		4: fbLinearAxis.AxisTargetPos := stStationPoses.rLinPosMotorPickup;
			OperatingState := E_OperatingState.MoveLinAxis;
			iOperatingStep := 5;
		5: MovePose(Pose := stStationPoses.aPoseLargeMotorPickupSt1,
				ExternalStatecontrol := 0,
				ExternalMove_ID := 0,
				Robot:= Meca500.GVL.Meca500, 
				Error=> Error, 
				Sent:= Sent, 
				Buffered:= Buffered);
		6: MoveLin(Pose := stStationPoses.aPoseLargeMotorPickupSt2,
				ExternalStatecontrol := 0,
				ExternalMove_ID := 0,
				Robot:= Meca500.GVL.Meca500, 
				Error=> Error, 
				Sent:= Sent, 
				Buffered:= Buffered);	
		7: SetCheckpoint(CheckpointID := 120,
				ExternalStatecontrol := 0,
				ExternalMove_ID := 0,
				Robot:= Meca500.GVL.Meca500, 
				Error=> Error, 
				Sent:= Sent, 
				Buffered:= Buffered);
		8: IF (stStationPoses.aPoseLargeMotorPickupSt2[1] + 20) < Meca500.GVL.Meca500.Inputs.End_Effector_Pose.SubIndex_001 THEN // If robot is closing on picking up motor but sensor is triggered, pause is flaged
				IF NOT stPlcCom.stPlcComIn.bRobotGripperSensor THEN
					Meca500.GVL.Meca500.Outputs.Motion_Control.Pause := TRUE;
					Meca500.GVL.Meca500.Outputs.Motion_Control.Clear_Move := TRUE;
					IF iWorkingStation <= 5 THEN
						PoseHome := PoseHome1;
					ELSE
						PoseHome := PoseHome2;
					END_IF
					Meca500.GVL.Meca500.Outputs.Motion_Control.Pause := FALSE;
					Meca500.GVL.Meca500.Outputs.Motion_Control.Clear_Move := FALSE;
					iOperatingStep := 9;
				END_IF
			ELSIF Meca500.GVL.Meca500.Inputs.Motion_Status.ReachedCheckPointId = 120 THEN
				IF NOT stPlcCom.stPlcComIn.bRobotGripperSensor THEN
					iOperatingStep := 12;
				ELSE
					IF iWorkingStation <= 5 THEN
						PoseHome := PoseHome1;
					ELSE
						PoseHome := PoseHome2;
					END_IF
					iOperatingStep := 9;
				END_IF
			END_IF
		9:  MoveLin(Pose := stStationPoses.aPoseLargeMotorPickupSt1,
				ExternalStatecontrol := 0,
				ExternalMove_ID := 0,
				Robot:= Meca500.GVL.Meca500, 
				Error=> Error, 
				Sent:= Sent, 
				Buffered:= Buffered);
		10:  MoveJoints(Joint_Angle := PoseHome,
				ExternalStatecontrol := 0,
				ExternalMove_ID := 0,
				Robot:= Meca500.GVL.Meca500, 
				Error=> Error, 
				Sent:= Sent, 
				Buffered:= Buffered);		
		11: DisableSetStation(iStationId := iWorkingStation);
			OperatingState := E_OperatingState.SetPoses;
			iOperatingStep := 0;
		12: MoveGripper(mm := 2,
				ExternalStatecontrol := 0,
				ExternalMove_ID := 0,
				Robot:= Meca500.GVL.Meca500, 
				Error=> Error, 
				Sent:= Sent, 
				Buffered:= Buffered);
		13: SetCheckpoint(CheckpointID := 101,
				ExternalStatecontrol := 0,
				ExternalMove_ID := 0,
				Robot:= Meca500.GVL.Meca500, 
				Error=> Error, 
				Sent:= Sent, 
				Buffered:= Buffered);
		14: IF Meca500.GVL.Meca500.Inputs.Motion_Status.ReachedCheckPointId = 101 AND EOAT[0] = 1 THEN
				IF EOAT[5] > 6.5 AND EOAT[5] < 7 AND NOT bMotorType THEN		
					iOperatingStep := 17;
				ELSE
					iOperatingStep := 15;
					bThicknessTestFailed := TRUE;
				END_IF
			END_IF
		15: MoveGripper(mm := 19,
				ExternalStatecontrol := 0,
				ExternalMove_ID := 0,
				Robot:= Meca500.GVL.Meca500, 
				Error=> Error, 
				Sent:= Sent, 
				Buffered:= Buffered);
		16: iOperatingStep := 9;
		17: MoveLin(Pose := stStationPoses.aPoseLargeMotorPickupSt3,
				ExternalStatecontrol := 0,
				ExternalMove_ID := 0,
				Robot:= Meca500.GVL.Meca500, 
				Error=> Error, 
				Sent:= Sent, 
				Buffered:= Buffered);
		18: SetCheckpoint(CheckpointID := 132,
				ExternalStatecontrol := 0,
				ExternalMove_ID := 0,
				Robot:= Meca500.GVL.Meca500, 
				Error=> Error, 
				Sent:= Sent, 
				Buffered:= Buffered);
		19: IF Meca500.GVL.Meca500.Inputs.Motion_Status.ReachedCheckPointId = 132 THEN
				iOperatingStep := 20;
			END_IF
		20: MovePose(Pose := PoseImagingGalvo14mm,
				ExternalStatecontrol := 0,
				ExternalMove_ID := 0,
				Robot:= Meca500.GVL.Meca500, 
				Error=> Error, 
				Sent:= Sent, 
				Buffered:= Buffered);	
		21: fbLinearAxis.AxisTargetPos := 40;
			OperatingState := E_OperatingState.MoveLinAxis;
			iOperatingStep := 22;
		22: SetCheckpoint(CheckpointID := 124,
				ExternalStatecontrol := 0,
				ExternalMove_ID := 0,
				Robot:= Meca500.GVL.Meca500, 
				Error=> Error, 
				Sent:= Sent, 
				Buffered:= Buffered);
		23: IF Meca500.GVL.Meca500.Inputs.Motion_Status.ReachedCheckPointId = 124 THEN
				iOperatingStep := 24;
			END_IF 
		24: stPlcCom.stPlcComOut.bRingLightGlue := TRUE;
			Trig.bMidStationCam := TRUE;
			iOperatingStep := 25;
		25: IF stCouplerData.bImagingDone THEN
				stPlcCom.stPlcComOut.bRingLightGlue := FALSE;
				Trig.bMidStationCam := FALSE;
				IF stCouplerData.bPartDetectSucceeded THEN
					stCouplerData.bImagingDone := FALSE;
					iOperatingStep := 26;
				ELSIF stCouplerData.bPartDetectFailed THEN
					stCouplerData.bImagingDone := FALSE;
					DisableSetStation(iStationId := iWorkingStation);					// LUO REJECT KÄYTÄNTÖ
					OperatingState := E_OperatingState.FinishedHandling14mm;
					iOperatingStep := 0;
				END_IF
			END_IF
		26:	fbLinearAxis.AxisTargetPos := 0;
			OperatingState := E_OperatingState.MoveLinAxis;
			iOperatingStep := 27;
		27: MovePose(Pose := PoseSafeInOutGlueSt1,
				ExternalStatecontrol := 0,
				ExternalMove_ID := 0,
				Robot:= Meca500.GVL.Meca500, 
				Error=> Error, 
				Sent:= Sent, 
				Buffered:= Buffered);	
		28: MoveJoints(Joint_Angle := PoseSafeInOutGlueSt2,
				ExternalStatecontrol := 0,
				ExternalMove_ID := 0,
				Robot:= Meca500.GVL.Meca500, 
				Error=> Error, 
				Sent:= Sent, 
				Buffered:= Buffered);	
		29: MoveLin(Pose := PoseSafeInOutGlueSt3,
				ExternalStatecontrol := 0,
				ExternalMove_ID := 0,
				Robot:= Meca500.GVL.Meca500, 
				Error=> Error, 
				Sent:= Sent, 
				Buffered:= Buffered);
		30: CheckType();
			iOperatingStep := 31;
		31: bBypassState := TRUE;
			 CASE iGluingStep OF
				0: stPlcCom.stPlcComOut.bGlueStopValve := TRUE;
					IF NOT stPlcCom.stPlcComIn.bGlueStopHome THEN
						MoveLin(Pose := PoseGluingSt1, // Pose To gluing
							ExternalStatecontrol := 0,
							ExternalMove_ID := 0,
							Robot:= Meca500.GVL.Meca500, 
							Error=> Error, 
							Sent:= Sent, 
							Buffered:= Buffered);				// LISÄÄ AJASTIN JOKA TARKISTAA ETTÄ VENTTIILI ON AUKI
					END_IF
				1: IF iGluingPoses = 5 THEN
						iGluingStep := 29;
					ELSE
						iGluingStep := 2;
					END_IF
				2:  MoveLin(Pose := PoseGluingSt2,  // NOTE!! LINEAR MOVEMENT Pose where gluing always has to start
						ExternalStatecontrol := 0,
						ExternalMove_ID := 0,
						Robot:= Meca500.GVL.Meca500, 
						Error=> Error, 
						Sent:= Sent, 
						Buffered:= Buffered);
				3: SetCartLinVel(
						Velocity_Limit := 0.4,
						ExternalStatecontrol := 0,
						ExternalMove_ID := 0,
						Robot:= Meca500.GVL.Meca500, 
						Error=> Error, 
						Sent:= Sent, 
						Buffered:= Buffered);
				4: SetCheckpoint(CheckpointID := 102,
						ExternalStatecontrol := 0,
						ExternalMove_ID := 0,
						Robot:= Meca500.GVL.Meca500, 
						Error=> Error, 
						Sent:= Sent, 
						Buffered:= Buffered);
				5: IF Meca500.GVL.Meca500.Inputs.Motion_Status.ReachedCheckPointId = 102 THEN
						stPlcCom.stPlcComOut.bTriggerGluing1 := TRUE;
						GluingStartTmr2.IN := TRUE;
						iGluingStep := 6;
					END_IF
				6: IF GluingStartTmr2.Q THEN
						GluingTmr2.IN := TRUE;
						GluingStartTmr2.IN := FALSE;
						iGluingStep := 7;
					END_IF
				7:  MoveLin(Pose := PoseGluingSt3,  // NOTE!! LINEAR MOVEMENT
						ExternalStatecontrol := 0,
						ExternalMove_ID := 0,
						Robot:= Meca500.GVL.Meca500, 
						Error=> Error, 
						Sent:= Sent, 
						Buffered:= Buffered);
				8: IF GluingTmr2.Q THEN
						stPlcCom.stPlcComOut.bTriggerGluing1 := FALSE;
						GluingTmr2.IN := FALSE;
						iGluingStep := 9;
					END_IF
				9: SetCheckpoint(CheckpointID := 104,
						ExternalStatecontrol := 0,
						ExternalMove_ID := 0,
						Robot:= Meca500.GVL.Meca500, 
						Error=> Error, 
						Sent:= Sent, 
						Buffered:= Buffered);
				10: IF Meca500.GVL.Meca500.Inputs.Motion_Status.ReachedCheckPointId = 104 THEN
						stPlcCom.stPlcComOut.bTriggerGluing1 := FALSE;
						IF iGluingPoses = 4 THEN
							iGluingStep := 11;
						ELSIF iGluingPoses = 3 THEN
							iGluingStep := 17;
						END_IF
					END_IF
				11: SetCartLinVel(
						Velocity_Limit := 10*rJogSpeed,
						ExternalStatecontrol := 0,
						ExternalMove_ID := 0,
						Robot:= Meca500.GVL.Meca500, 
						Error=> Error, 
						Sent:= Sent, 
						Buffered:= Buffered);
				12: MoveLin(Pose := PoseGluingSt1,  // NOTE!! LINEAR MOVEMENT
						ExternalStatecontrol := 0,
						ExternalMove_ID := 0,
						Robot:= Meca500.GVL.Meca500, 
						Error=> Error, 
						Sent:= Sent, 
						Buffered:= Buffered);
				13: MoveLin(Pose := PoseGluingSt4,  // NOTE!! LINEAR MOVEMENT
						ExternalStatecontrol := 0,
						ExternalMove_ID := 0,
						Robot:= Meca500.GVL.Meca500, 
						Error=> Error, 
						Sent:= Sent, 
						Buffered:= Buffered);
				14: SetCheckpoint(CheckpointID := 105,
						ExternalStatecontrol := 0,
						ExternalMove_ID := 0,
						Robot:= Meca500.GVL.Meca500, 
						Error=> Error, 
						Sent:= Sent, 
						Buffered:= Buffered);
				15: IF Meca500.GVL.Meca500.Inputs.Motion_Status.ReachedCheckPointId = 105 THEN
						stPlcCom.stPlcComOut.bTriggerGluing1 := TRUE;
						GluingTmr1.IN := TRUE;
						iGluingStep := 16;
					END_IF
				16: IF GluingTmr1.Q THEN
						GluingTmr1.IN := FALSE;
						iGluingStep := 17;
						stPlcCom.stPlcComOut.bTriggerGluing1 := FALSE;
					END_IF
				17:  SetCartLinVel(
						Velocity_Limit := 10*rJogSpeed,
						ExternalStatecontrol := 0,
						ExternalMove_ID := 0,
						Robot:= Meca500.GVL.Meca500, 
						Error=> Error, 
						Sent:= Sent, 
						Buffered:= Buffered);
				18:  MoveLin(Pose := PoseGluingSt1,  // NOTE!! LINEAR MOVEMENT
						ExternalStatecontrol := 0,
						ExternalMove_ID := 0,
						Robot:= Meca500.GVL.Meca500, 
						Error=> Error, 
						Sent:= Sent, 
						Buffered:= Buffered);
				19: SetCheckpoint(CheckpointID := 106,
						ExternalStatecontrol := 0,
						ExternalMove_ID := 0,
						Robot:= Meca500.GVL.Meca500, 
						Error=> Error, 
						Sent:= Sent, 
						Buffered:= Buffered);
				
				20: IF Meca500.GVL.Meca500.Inputs.Motion_Status.ReachedCheckPointId = 106 THEN
						stPlcCom.stPlcComOut.bTriggerGluing1 := FALSE;
						GluingTmr1.IN := FALSE;
						iGluingStep := 41;
					END_IF
				29:  SetCartLinVel(
						Velocity_Limit := 0.4,
						ExternalStatecontrol := 0,
						ExternalMove_ID := 0,
						Robot:= Meca500.GVL.Meca500, 
						Error=> Error, 
						Sent:= Sent, 
						Buffered:= Buffered);
				30: MoveLin(Pose := PoseGluingSt2,  // NOTE!! LINEAR MOVEMENT Pose where gluing always has to start
						ExternalStatecontrol := 0,
						ExternalMove_ID := 0,
						Robot:= Meca500.GVL.Meca500, 
						Error=> Error, 
						Sent:= Sent, 
						Buffered:= Buffered);
				31: SetCheckpoint(CheckpointID := 102,
						ExternalStatecontrol := 0,
						ExternalMove_ID := 0,
						Robot:= Meca500.GVL.Meca500, 
						Error=> Error, 
						Sent:= Sent, 
						Buffered:= Buffered);
				32: IF Meca500.GVL.Meca500.Inputs.Motion_Status.ReachedCheckPointId = 102 THEN
						stPlcCom.stPlcComOut.bTriggerGluing1 := TRUE;
						iGluingStep := 33;
					END_IF
				33:  MoveLin(Pose := PoseGluingSt3,  // NOTE!! LINEAR MOVEMENT Pose where gluing always has to start
						ExternalStatecontrol := 0,
						ExternalMove_ID := 0,
						Robot:= Meca500.GVL.Meca500, 
						Error=> Error, 
						Sent:= Sent, 
						Buffered:= Buffered);
				34: MoveLin(Pose := PoseGluingSt4,  // NOTE!! LINEAR MOVEMENT Pose where gluing always has to start
						ExternalStatecontrol := 0,
						ExternalMove_ID := 0,
						Robot:= Meca500.GVL.Meca500, 
						Error=> Error, 
						Sent:= Sent, 
						Buffered:= Buffered);
				35: MoveLin(Pose := PoseGluingSt5,  // NOTE!! LINEAR MOVEMENT Pose where gluing always has to start
						ExternalStatecontrol := 0,
						ExternalMove_ID := 0,
						Robot:= Meca500.GVL.Meca500, 
						Error=> Error, 
						Sent:= Sent, 
						Buffered:= Buffered);
				36: SetCheckpoint(CheckpointID := 109,
						ExternalStatecontrol := 0,
						ExternalMove_ID := 0,
						Robot:= Meca500.GVL.Meca500, 
						Error=> Error, 
						Sent:= Sent, 
						Buffered:= Buffered);
				37: IF Meca500.GVL.Meca500.Inputs.Motion_Status.ReachedCheckPointId = 109 THEN
						stPlcCom.stPlcComOut.bTriggerGluing1 := FALSE;
						iGluingStep := 38;
					END_IF
				38: MoveLin(Pose := PoseGluingSt1,  // NOTE!! LINEAR MOVEMENT Pose where gluing always has to start
						ExternalStatecontrol := 0,
						ExternalMove_ID := 0,
						Robot:= Meca500.GVL.Meca500, 
						Error=> Error, 
						Sent:= Sent, 
						Buffered:= Buffered);	
				39: SetCartLinVel(
						Velocity_Limit := 10*rJogSpeed,
						ExternalStatecontrol := 0,
						ExternalMove_ID := 0,
						Robot:= Meca500.GVL.Meca500, 
						Error=> Error, 
						Sent:= Sent, 
						Buffered:= Buffered);
						
				40: SetCheckpoint(CheckpointID := 106,
						ExternalStatecontrol := 0,
						ExternalMove_ID := 0,
						Robot:= Meca500.GVL.Meca500, 
						Error=> Error, 
						Sent:= Sent, 
						Buffered:= Buffered);
				41: IF Meca500.GVL.Meca500.Inputs.Motion_Status.ReachedCheckPointId = 106 THEN
						stPlcCom.stPlcComOut.bTriggerGluing1 := FALSE;
						stPlcCom.stPlcComOut.bGlueStopValve := FALSE;
						bBypassState := FALSE;
						iOperatingStep := 32;
						iGluingStep := 0;
					END_IF
			END_CASE
			IF Sent AND Buffered AND bBypassState THEN
				iGluingStep := iGluingStep +1;
				Sent := FALSE;
				Buffered := FALSE;
			END_IF

		32:  MoveLin(Pose := PoseSafeInOutGlueSt3,
				ExternalStatecontrol := 0,
				ExternalMove_ID := 0,
				Robot:= Meca500.GVL.Meca500, 
				Error=> Error, 
				Sent:= Sent, 
				Buffered:= Buffered);
		33: MoveJoints(Joint_Angle := PoseSafeInOutGlueSt2,
				ExternalStatecontrol := 0,
				ExternalMove_ID := 0,
				Robot:= Meca500.GVL.Meca500, 
				Error=> Error, 
				Sent:= Sent, 
				Buffered:= Buffered);
		34: MovePose(Pose := PoseSafeInOutGlueSt1,
				ExternalStatecontrol := 0,
				ExternalMove_ID := 0,
				Robot:= Meca500.GVL.Meca500, 
				Error=> Error, 
				Sent:= Sent, 
				Buffered:= Buffered);
		35: MoveJoints(Joint_Angle := PoseAfterGluingSt1,
				ExternalStatecontrol := 0,
				ExternalMove_ID := 0,
				Robot:= Meca500.GVL.Meca500, 
				Error=> Error, 
				Sent:= Sent, 
				Buffered:= Buffered);
		36:  fbLinearAxis.AxisTargetPos := stStationPoses.rLinPosPlace;
			OperatingState := E_OperatingState.MoveLinAxis;
			iOperatingStep := 37;
			stStationPoses.aPoseLargeMotorPlaceSt2[5] := stStationPoses.aPoseLargeMotorPlaceSt2[5] - (stCouplerData.rCouplerAngleDeg);
		37: MovePose(Pose := stStationPoses.aPoseLargeMotorPlaceSt1,
				ExternalStatecontrol := 0,
				ExternalMove_ID := 0,
				Robot:= Meca500.GVL.Meca500, 
				Error=> Error, 
				Sent:= Sent, 
				Buffered:= Buffered);
		38: MoveLin(Pose := stStationPoses.aPoseLargeMotorPlaceSt2,
				ExternalStatecontrol := 0,
				ExternalMove_ID := 0,
				Robot:= Meca500.GVL.Meca500, 
				Error=> Error, 
				Sent:= Sent, 
				Buffered:= Buffered);	
		39: SetCheckpoint(CheckpointID := 104,
				ExternalStatecontrol := 0,
				ExternalMove_ID := 0,
				Robot:= Meca500.GVL.Meca500, 
				Error=> Error, 
				Sent:= Sent, 
				Buffered:= Buffered);
		
		40: IF Meca500.GVL.Meca500.Inputs.Motion_Status.ReachedCheckPointId = 104 THEN
				EngageHolder();
				StationGripperTmr.IN := TRUE;
				IF StationGripperTmr.Q AND bHolderSensor THEN
					StationGripperTmr.IN := FALSE;
					stStationPoses.aPoseLargeMotorPlaceSt2[5] := 0;
					iOperatingStep := 41;
				END_IF
			END_IF
		41: MoveGripper(mm := 20,
				ExternalStatecontrol := 0,
				ExternalMove_ID := 0,
				Robot:= Meca500.GVL.Meca500, 
				Error=> Error, 
				Sent:= Sent, 
				Buffered:= Buffered);
		42: IF EOAT[1] = 1 AND EOAT[0] = 0 THEN
				MoveLin(Pose := stStationPoses.aPoseLargeMotorPlaceSt2,
					ExternalStatecontrol := 0,
					ExternalMove_ID := 0,
					Robot:= Meca500.GVL.Meca500, 
					Error=> Error, 
					Sent:= Sent, 
					Buffered:= Buffered);
// 					iOperatingStep := 43;
			END_IF
		43: MovePose(Pose := stStationPoses.aPoseLargeMotorPlaceSt3,
				ExternalStatecontrol := 0,
				ExternalMove_ID := 0,
				Robot:= Meca500.GVL.Meca500, 
				Error=> Error, 
				Sent:= Sent, 
				Buffered:= Buffered);
		44: SetTrf(
				Pose := PoseTRFMirror,
				ExternalStatecontrol := 0,
				ExternalMove_ID := 0,
				Robot:= Meca500.GVL.Meca500, 
				Error=> Error, 
				Sent:= Sent, 
				Buffered:= Buffered);
		45: MoveJoints(Joint_Angle := PoseToMirrorPickupSt1,
				ExternalStatecontrol := 0,
				ExternalMove_ID := 0,
				Robot:= Meca500.GVL.Meca500, 
				Error=> Error, 
				Sent:= Sent, 
				Buffered:= Buffered);
		46: fbLinearAxis.AxisTargetPos := stStationPoses.rLinPosMirrorPickup;
			OperatingState := E_OperatingState.MoveLinAxis;
			iOperatingStep := 47;
		47: MoveGripper(mm := 21,
				ExternalStatecontrol := 0,
				ExternalMove_ID := 0,
				Robot:= Meca500.GVL.Meca500, 
				Error=> Error, 
				Sent:= Sent, 
				Buffered:= Buffered);
		48: SetGripperForce(
				Force := 5,
				ExternalStatecontrol := 0,
				ExternalMove_ID := 0,
				Robot:= Meca500.GVL.Meca500, 
				Error=> Error, 
				Sent:= Sent, 
				Buffered:= Buffered);
		49: MovePose(Pose := stStationPoses.aPoseMirrorPickupSt1,
				ExternalStatecontrol := 0,
				ExternalMove_ID := 0,
				Robot:= Meca500.GVL.Meca500, 
				Error=> Error, 
				Sent:= Sent, 
				Buffered:= Buffered);
		50: MovePose(Pose := stStationPoses.aPoseMirrorPickupSt2,
				ExternalStatecontrol := 0,
				ExternalMove_ID := 0,
				Robot:= Meca500.GVL.Meca500, 
				Error=> Error, 
				Sent:= Sent, 
				Buffered:= Buffered);
		51: MoveGripper(mm := 8,
				ExternalStatecontrol := 0,
				ExternalMove_ID := 0,
				Robot:= Meca500.GVL.Meca500, 
				Error=> Error, 
				Sent:= Sent, 
				Buffered:= Buffered);
		52: IF EOAT[0] = 1 THEN
				iOperatingStep := 53;
			END_IF
		53: MovePose(Pose := stStationPoses.aPoseMirrorPickupSt1,
				ExternalStatecontrol := 0,
				ExternalMove_ID := 0,
				Robot:= Meca500.GVL.Meca500, 
				Error=> Error, 
				Sent:= Sent, 
				Buffered:= Buffered);
		54: SetCheckpoint(CheckpointID := 109,
				ExternalStatecontrol := 0,
				ExternalMove_ID := 0,
				Robot:= Meca500.GVL.Meca500, 
				Error=> Error, 
				Sent:= Sent, 
				Buffered:= Buffered);
		55: IF Meca500.GVL.Meca500.Inputs.Motion_Status.ReachedCheckPointId = 109 THEN
				iOperatingStep := 56;
			END_IF
		56: fbLinearAxis.AxisTargetPos := stStationPoses.rLinPosPlace;
			OperatingState := E_OperatingState.MoveLinAxis;
			iOperatingStep := 57;
		57: MovePose(Pose := stStationPoses.aPoseMirrorPlaceSt1,
				ExternalStatecontrol := 0,
				ExternalMove_ID := 0,
				Robot:= Meca500.GVL.Meca500, 
				Error=> Error, 
				Sent:= Sent, 
				Buffered:= Buffered);
		58: MoveLin(Pose := stStationPoses.aPoseMirrorPlaceSt2,
				ExternalStatecontrol := 0,
				ExternalMove_ID := 0,
				Robot:= Meca500.GVL.Meca500, 
				Error=> Error, 
				Sent:= Sent, 
				Buffered:= Buffered);
		59: SetCartLinVel(
				Velocity_Limit := 1,
				ExternalStatecontrol := 0,
				ExternalMove_ID := 0,
				Robot:= Meca500.GVL.Meca500, 
				Error=> Error, 
				Sent:= Sent, 
				Buffered:= Buffered);
		60: MoveLin(Pose := stStationPoses.aPoseMirrorPlaceSt3,
				ExternalStatecontrol := 0,
				ExternalMove_ID := 0,
				Robot:= Meca500.GVL.Meca500, 
				Error=> Error, 
				Sent:= Sent, 
				Buffered:= Buffered);
		61: SetCheckpoint(CheckpointID := 107,
				ExternalStatecontrol := 0,
				ExternalMove_ID := 0,
				Robot:= Meca500.GVL.Meca500, 
				Error=> Error, 
				Sent:= Sent, 
				Buffered:= Buffered);
		
		62: IF Meca500.GVL.Meca500.Inputs.Motion_Status.ReachedCheckPointId = 107 THEN
				EngageSlider();
				stStationPoses.aPoseMirrorPlaceSt1[1] := stStationPoses.aPoseMirrorPlaceSt3[1];
				stStationPoses.aPoseMirrorPlaceSt1[2] := stStationPoses.aPoseMirrorPlaceSt3[2];
				StationGripperTmr.IN := TRUE;
				IF StationGripperTmr.Q AND NOT bSliderSensor THEN
					StationGripperTmr.IN := FALSE;
					iOperatingStep := 63;
				END_IF
			END_IF
		63: MoveGripper(mm := 21,
				ExternalStatecontrol := 0,
				ExternalMove_ID := 0,
				Robot:= Meca500.GVL.Meca500, 
				Error=> Error, 
				Sent:= Sent, 
				Buffered:= Buffered);
		64: SetCartLinVel(
				Velocity_Limit := 10*rJogSpeed,
				ExternalStatecontrol := 0,
				ExternalMove_ID := 0,
				Robot:= Meca500.GVL.Meca500, 
				Error=> Error, 
				Sent:= Sent, 
				Buffered:= Buffered);
		65: MovePose(Pose := stStationPoses.aPoseMirrorPlaceSt1,
				ExternalStatecontrol := 0,
				ExternalMove_ID := 0,
				Robot:= Meca500.GVL.Meca500, 
				Error=> Error, 
				Sent:= Sent, 
				Buffered:= Buffered);
		66: MoveJoints(Joint_Angle := PoseHome2,
				ExternalStatecontrol := 0,
				ExternalMove_ID := 0,
				Robot:= Meca500.GVL.Meca500, 
				Error=> Error, 
				Sent:= Sent, 
				Buffered:= Buffered);
		67: OperatingState := E_OperatingState.SetPoses;
			iOperatingStep := 0;
		100:  MoveLin(Pose := stStationPoses.aPoseLargeMotorPickupSt1,
				ExternalStatecontrol := 0,
				ExternalMove_ID := 0,
				Robot:= Meca500.GVL.Meca500, 
				Error=> Error, 
				Sent:= Sent, 
				Buffered:= Buffered);
		101: MovePose(Pose := PoseHome,
				ExternalStatecontrol := 0,
				ExternalMove_ID := 0,
				Robot:= Meca500.GVL.Meca500, 
				Error=> Error, 
				Sent:= Sent, 
				Buffered:= Buffered);
		102: MoveGripper(mm := 24,
				ExternalStatecontrol := 0,
				ExternalMove_ID := 0,
				Robot:= Meca500.GVL.Meca500, 
				Error=> Error, 
				Sent:= Sent, 
				Buffered:= Buffered);
		103: SetCheckpoint(CheckpointID := 1000,
				ExternalStatecontrol := 0,
				ExternalMove_ID := 0,
				Robot:= Meca500.GVL.Meca500, 
				Error=> Error, 
				Sent:= Sent, 
				Buffered:= Buffered);
		104: IF Meca500.GVL.Meca500.Inputs.Motion_Status.ReachedCheckPointId = 1000 THEN
				bRobotHomed := TRUE;
				iOperatingStep := 0;
			END_IF
END_CASE
IF Sent AND Buffered AND NOT bBypassState THEN
	iOperatingStep := iOperatingStep +1;
	Sent := FALSE;
	Buffered := FALSE;
END_IF
END_ACTION

METHOD Initialize : BOOL
VAR_INPUT
END_VAR

iOperatingStep := 0;
Sent := FALSE;
Buffered := FALSE;
GluingTmr1.IN := FALSE;
GluingTmr2.IN := FALSE;
GluingOffTmr.IN := FALSE;
GluingStartTmr2.IN := FALSE;
StationGripperTmr.IN := FALSE;
eCurrentState := E_CurrentState.Init;
ReleaseTmr.IN := FALSE;
StationGripperTmr.IN :=FALSE;
iMirrorStep := 0;
iFinishedStep := 0;
bDismountingActive := FALSE;
END_METHOD

ACTION MirrorAdj:
eCurrentState := E_CurrentState.MirrorAdj;
bOperatingActive := TRUE;
CASE iMirrorStep OF
	0: MoveGripper(mm := 20,
			ExternalStatecontrol := 0,
			ExternalMove_ID := 0,
			Robot:= Meca500.GVL.Meca500, 
			Error=> Error, 
			Sent:= Sent, 
			Buffered:= Buffered);
	1: IF EOAT[1] = 1 AND EOAT[0] = 0 THEN
			IF iWorkingStation < 5 THEN
				iMirrorStep := 2;
			ELSE
				iMirrorStep := 4;
			END_IF
			
		END_IF
	2: MoveJoints(Joint_Angle := PoseHome2,
			ExternalStatecontrol := 0,
			ExternalMove_ID := 0,
			Robot:= Meca500.GVL.Meca500, 
			Error=> Error, 
			Sent:= Sent, 
			Buffered:= Buffered);
	3: iMirrorStep := 5;
	4: MoveJoints(Joint_Angle := PoseHome1,
			ExternalStatecontrol := 0,
			ExternalMove_ID := 0,
			Robot:= Meca500.GVL.Meca500, 
			Error=> Error, 
			Sent:= Sent, 
			Buffered:= Buffered);
	5: SetCheckpoint(CheckpointID := 15,
			ExternalStatecontrol := 0,
			ExternalMove_ID := 0,
			Robot:= Meca500.GVL.Meca500, 
			Error=> Error, 
			Sent:= Sent, 
			Buffered:= Buffered);
	6: IF Meca500.GVL.Meca500.Inputs.Motion_Status.ReachedCheckPointId = 15 THEN
		SetAdjustmentPoses();
			 SetTrf(
				Pose := PoseTRFMirror,
				ExternalStatecontrol := 0,
				ExternalMove_ID := 0,
				Robot:= Meca500.GVL.Meca500, 
				Error=> Error, 
				Sent:= Sent, 
				Buffered:= Buffered);
		END_IF
	7:  fbLinearAxis.AxisTargetPos := stStationPoses.rLinPosPlace;
		OperatingState := E_OperatingState.MoveLinAxis;
		iMirrorStep := 8;
	8:	SetGripperForce(
			Force := 5,
			ExternalStatecontrol := 0,
			ExternalMove_ID := 0,
			Robot:= Meca500.GVL.Meca500, 
			Error=> Error, 
			Sent:= Sent, 
			Buffered:= Buffered);
	9: MoveLin(Pose := stStationPoses.aPoseMirrorPlaceSt1,
			ExternalStatecontrol := 0,
			ExternalMove_ID := 0,
			Robot:= Meca500.GVL.Meca500, 
			Error=> Error, 
			Sent:= Sent, 
			Buffered:= Buffered);
	10: MoveLin(Pose := PoseMirrorAdjustPrev,
			ExternalStatecontrol := 0,
			ExternalMove_ID := 0,
			Robot:= Meca500.GVL.Meca500, 
			Error=> Error, 
			Sent:= Sent, 
			Buffered:= Buffered);
	11: MoveGripper(mm := 0,
			ExternalStatecontrol := 0,
			ExternalMove_ID := 0,
			Robot:= Meca500.GVL.Meca500, 
			Error=> Error, 
			Sent:= Sent, 
			Buffered:= Buffered);
	12:SetCartLinVel(
			Velocity_Limit := 5,
			ExternalStatecontrol := 0,
			ExternalMove_ID := 0,
			Robot:= Meca500.GVL.Meca500, 
			Error=> Error, 
			Sent:= Sent, 
			Buffered:= Buffered);
	13: IF EOAT[0] = 1 THEN
			iMirrorStep := 14;
		END_IF
	14: MoveLin(Pose := PoseMirrorAdjust,
			ExternalStatecontrol := 0,
			ExternalMove_ID := 0,
			Robot:= Meca500.GVL.Meca500, 
			Error=> Error, 
			Sent:= Sent, 
			Buffered:= Buffered);
	15: SetCheckpoint(CheckpointID := 16,
			ExternalStatecontrol := 0,
			ExternalMove_ID := 0,
			Robot:= Meca500.GVL.Meca500, 
			Error=> Error, 
			Sent:= Sent, 
			Buffered:= Buffered);
	16: IF Meca500.GVL.Meca500.Inputs.Motion_Status.ReachedCheckPointId = 16 THEN
			iMirrorStep := 17;
		END_IF
	17: MoveGripper(mm := 20,
			ExternalStatecontrol := 0,
			ExternalMove_ID := 0,
			Robot:= Meca500.GVL.Meca500, 
			Error=> Error, 
			Sent:= Sent, 
			Buffered:= Buffered);
	18: SetCartLinVel(
			Velocity_Limit := 10*rJogSpeed,
			ExternalStatecontrol := 0,
			ExternalMove_ID := 0,
			Robot:= Meca500.GVL.Meca500, 
			Error=> Error, 
			Sent:= Sent, 
			Buffered:= Buffered);
	19: IF EOAT[0] = 0 THEN
			iMirrorStep := 20;
		END_IF
	20: MoveLin(Pose := stStationPoses.aPoseMirrorPlaceSt1,
			ExternalStatecontrol := 0,
			ExternalMove_ID := 0,
			Robot:= Meca500.GVL.Meca500, 
			Error=> Error, 
			Sent:= Sent, 
			Buffered:= Buffered);
	21: IF iWorkingStation < 5 THEN
			iMirrorStep := 22;
		ELSE
			iMirrorStep := 23;
		END_IF
	22: MoveJoints(Joint_Angle := PoseHome2,
			ExternalStatecontrol := 0,
			ExternalMove_ID := 0,
			Robot:= Meca500.GVL.Meca500, 
			Error=> Error, 
			Sent:= Sent, 
			Buffered:= Buffered);
	23: iMirrorStep := 25;
	24: MoveJoints(Joint_Angle := PoseHome1,
			ExternalStatecontrol := 0,
			ExternalMove_ID := 0,
			Robot:= Meca500.GVL.Meca500, 
			Error=> Error, 
			Sent:= Sent, 
			Buffered:= Buffered);
	
	25: SetCheckpoint(CheckpointID := 17,
			ExternalStatecontrol := 0,
			ExternalMove_ID := 0,
			Robot:= Meca500.GVL.Meca500, 
			Error=> Error, 
			Sent:= Sent, 
			Buffered:= Buffered);
	26: IF Meca500.GVL.Meca500.Inputs.Motion_Status.ReachedCheckPointId = 17 THEN
			AdjDone();
			iMirrorStep := 0;
			OperatingState := E_OperatingState.SetPoses;
		END_IF
END_CASE
IF Sent AND Buffered THEN
	iMirrorStep := iMirrorStep +1;
	Sent := FALSE;
	Buffered := FALSE;
END_IF
END_ACTION

METHOD MirrorOffset : BOOL
VAR_INPUT
END_VAR
CASE iWorkingStation OF
	1..5: stStationPoses.aPoseMirrorPlaceSt2[1] := stStationPoses.aPoseMirrorPlaceSt2[1] + stAssemblyData.Station1To5.rMirrorCenterOffsetToWeightCenterY; 
		stStationPoses.aPoseMirrorPlaceSt3[1] := stStationPoses.aPoseMirrorPlaceSt3[1] + stAssemblyData.Station1To5.rMirrorCenterOffsetToWeightCenterY;
	6..10: stStationPoses.aPoseMirrorPlaceSt2[1] := stStationPoses.aPoseMirrorPlaceSt2[1] + stAssemblyData.Station5To10.rMirrorCenterOffsetToWeightCenterY; 
		stStationPoses.aPoseMirrorPlaceSt3[1] := stStationPoses.aPoseMirrorPlaceSt3[1] + stAssemblyData.Station5To10.rMirrorCenterOffsetToWeightCenterY;
END_CASE
END_METHOD

METHOD ReleaseHolder : BOOL
VAR_INPUT
END_VAR
CASE iWorkingStation OF
	0: 
	1: stStation.fbSts1.bEngageHolder := FALSE;
		IF stStation.fbSts1.bHolderSensor THEN
			bHolderSensor := TRUE;
		ELSE
			bHolderSensor := FALSE;
		END_IF
	2: stStation.fbSts2.bEngageHolder := FALSE;
		IF stStation.fbSts2.bHolderSensor THEN
			bHolderSensor := TRUE;
		ELSE
			bHolderSensor := FALSE;
		END_IF
	3: stStation.fbSts3.bEngageHolder := FALSE;
		IF stStation.fbSts3.bHolderSensor THEN
			bHolderSensor := TRUE;
		ELSE
			bHolderSensor := FALSE;
		END_IF
	4: stStation.fbSts4.bEngageHolder := FALSE;
		IF stStation.fbSts4.bHolderSensor THEN
			bHolderSensor := TRUE;
		ELSE
			bHolderSensor := FALSE;
		END_IF
	5: stStation.fbSts5.bEngageHolder := FALSE;
		IF stStation.fbSts5.bHolderSensor THEN
			bHolderSensor := TRUE;
		ELSE
			bHolderSensor := FALSE;
		END_IF
	6: stStation.fbSts6.bEngageHolder := FALSE;
		IF stStation.fbSts6.bHolderSensor THEN
			bHolderSensor := TRUE;
		ELSE
			bHolderSensor := FALSE;
		END_IF
	7: stStation.fbSts7.bEngageHolder := FALSE;
		IF stStation.fbSts7.bHolderSensor THEN
			bHolderSensor := TRUE;
		ELSE
			bHolderSensor := FALSE;
		END_IF
	8: stStation.fbSts8.bEngageHolder := FALSE;
		IF stStation.fbSts8.bHolderSensor THEN
			bHolderSensor := TRUE;
		ELSE
			bHolderSensor := FALSE;
		END_IF
	9: stStation.fbSts9.bEngageHolder := FALSE;
		IF stStation.fbSts9.bHolderSensor THEN
			bHolderSensor := TRUE;
		ELSE
			bHolderSensor := FALSE;
		END_IF
	10: stStation.fbSts10.bEngageHolder := FALSE;
		IF stStation.fbSts10.bHolderSensor THEN
			bHolderSensor := TRUE;
		ELSE
			bHolderSensor := FALSE;
		END_IF
END_CASE
END_METHOD

METHOD ReleaseSlider : BOOL
VAR_INPUT
END_VAR
CASE iWorkingStation OF
	0: 
	1: stStation.fbSts1.bEngageSlider := FALSE;
		IF stStation.fbSts1.bSliderSensor THEN
			bSliderSensor := FALSE;
		ELSE
			bSliderSensor := TRUE;
		END_IF
	2: stStation.fbSts2.bEngageSlider := FALSE;
		IF stStation.fbSts2.bSliderSensor THEN
			bSliderSensor := FALSE;
		ELSE
			bSliderSensor := TRUE;
		END_IF
	3: stStation.fbSts3.bEngageSlider := FALSE;
		IF stStation.fbSts3.bSliderSensor THEN
			bSliderSensor := FALSE;
		ELSE
			bSliderSensor := TRUE;
		END_IF
	4: stStation.fbSts4.bEngageSlider := FALSE;
		IF stStation.fbSts4.bSliderSensor THEN
			bSliderSensor := FALSE;
		ELSE
			bSliderSensor := TRUE;
		END_IF
	5: stStation.fbSts5.bEngageSlider := FALSE;
		IF stStation.fbSts5.bSliderSensor THEN
			bSliderSensor := FALSE;
		ELSE
			bSliderSensor := TRUE;
		END_IF
	6: stStation.fbSts6.bEngageSlider := FALSE;
		IF stStation.fbSts6.bSliderSensor THEN
			bSliderSensor := FALSE;
		ELSE
			bSliderSensor := TRUE;
		END_IF
	7: stStation.fbSts7.bEngageSlider := FALSE;
		IF stStation.fbSts7.bSliderSensor THEN
			bSliderSensor := FALSE;
		ELSE
			bSliderSensor := TRUE;
		END_IF
	8: stStation.fbSts8.bEngageSlider := FALSE;
		IF stStation.fbSts8.bSliderSensor THEN
			bSliderSensor := FALSE;
		ELSE
			bSliderSensor := TRUE;
		END_IF
	9: stStation.fbSts9.bEngageSlider := FALSE;
		IF stStation.fbSts9.bSliderSensor THEN
			bSliderSensor := FALSE;
		ELSE
			bSliderSensor := TRUE;
		END_IF
	10: stStation.fbSts10.bEngageSlider := FALSE;
		IF stStation.fbSts10.bSliderSensor THEN
			bSliderSensor := FALSE;
		ELSE
			bSliderSensor := TRUE;
		END_IF
END_CASE
END_METHOD

METHOD SetAdjustmentPoses : BOOL
VAR_INPUT
END_VAR
CASE iWorkingStation OF
	1: IF stStation.fbSts1.iAdjustmentCount < 1 THEN
			PoseMirrorAdjustPrev  := stStationPoses.aPoseMirrorPlaceSt3;
			PoseMirrorAdjust := stStationPoses.aPoseMirrorPlaceSt3;
			PoseMirrorAdjust[1] := stStationPoses.aPoseMirrorPlaceSt3[1] + stStation.fbSts1.rRobotAdjValue;

		ELSE
			PoseMirrorAdjustPrev := PoseMirrorAdjustPrevSts1;
			PoseMirrorAdjust := PoseMirrorAdjustPrevSts1;
			PoseMirrorAdjust[1] := PoseMirrorAdjustPrevSts1[1] + stStation.fbSts1.rRobotAdjValue;
		END_IF
	2: IF stStation.fbSts2.iAdjustmentCount < 1 THEN
			PoseMirrorAdjustPrev  := stStationPoses.aPoseMirrorPlaceSt3;
			PoseMirrorAdjust := stStationPoses.aPoseMirrorPlaceSt3;
			PoseMirrorAdjust[1] := stStationPoses.aPoseMirrorPlaceSt3[1] + stStation.fbSts2.rRobotAdjValue;
		ELSE
			PoseMirrorAdjustPrev := PoseMirrorAdjustPrevSts2;
			PoseMirrorAdjust := PoseMirrorAdjustPrevSts2;
			PoseMirrorAdjust[1] := PoseMirrorAdjustPrevSts2[1] + stStation.fbSts2.rRobotAdjValue;
		END_IF
		
	3:  IF stStation.fbSts3.iAdjustmentCount < 1 THEN
			PoseMirrorAdjustPrev  := stStationPoses.aPoseMirrorPlaceSt3;
			PoseMirrorAdjust := stStationPoses.aPoseMirrorPlaceSt3;
			PoseMirrorAdjust[2] := stStationPoses.aPoseMirrorPlaceSt3[2] + stStation.fbSts3.rRobotAdjValue;
		ELSE
			PoseMirrorAdjustPrev := PoseMirrorAdjustPrevSts3;
			PoseMirrorAdjust := PoseMirrorAdjustPrevSts3;
			PoseMirrorAdjust[2] := PoseMirrorAdjustPrevSts3[2] - stStation.fbSts3.rRobotAdjValue;
		END_IF
	4:  IF stStation.fbSts4.iAdjustmentCount < 1 THEN
			PoseMirrorAdjustPrev  := stStationPoses.aPoseMirrorPlaceSt3;
			PoseMirrorAdjust := stStationPoses.aPoseMirrorPlaceSt3;
			PoseMirrorAdjust[2] := stStationPoses.aPoseMirrorPlaceSt3[2] + stStation.fbSts4.rRobotAdjValue;
		ELSE
			PoseMirrorAdjustPrev := PoseMirrorAdjustPrevSts4;
			PoseMirrorAdjust := PoseMirrorAdjustPrevSts4;
			PoseMirrorAdjust[2] := PoseMirrorAdjustPrevSts4[2] - stStation.fbSts4.rRobotAdjValue;
		END_IF
	5:  IF stStation.fbSts5.iAdjustmentCount < 1 THEN
			PoseMirrorAdjustPrev  := stStationPoses.aPoseMirrorPlaceSt3;
			PoseMirrorAdjust := stStationPoses.aPoseMirrorPlaceSt3;
			PoseMirrorAdjust[2] := stStationPoses.aPoseMirrorPlaceSt3[2] + stStation.fbSts5.rRobotAdjValue;
		ELSE
			PoseMirrorAdjustPrev := PoseMirrorAdjustPrevSts5;
			PoseMirrorAdjust := PoseMirrorAdjustPrevSts5;
			PoseMirrorAdjust[2] := PoseMirrorAdjustPrevSts5[2] - stStation.fbSts5.rRobotAdjValue;
		END_IF
	6:  IF stStation.fbSts6.iAdjustmentCount < 1 THEN
			PoseMirrorAdjustPrev  := stStationPoses.aPoseMirrorPlaceSt3;
			PoseMirrorAdjust := stStationPoses.aPoseMirrorPlaceSt3;
			PoseMirrorAdjust[2] := stStationPoses.aPoseMirrorPlaceSt3[2] + stStation.fbSts6.rRobotAdjValue;
		ELSE
			PoseMirrorAdjustPrev := PoseMirrorAdjustPrevSts6;
			PoseMirrorAdjust := PoseMirrorAdjustPrevSts6;
			PoseMirrorAdjust[2] := PoseMirrorAdjustPrevSts6[2] - stStation.fbSts6.rRobotAdjValue;
		END_IF
	7: IF stStation.fbSts7.iAdjustmentCount < 1 THEN
			PoseMirrorAdjustPrev  := stStationPoses.aPoseMirrorPlaceSt3;
			PoseMirrorAdjust := stStationPoses.aPoseMirrorPlaceSt3;
			PoseMirrorAdjust[2] := stStationPoses.aPoseMirrorPlaceSt3[2] + stStation.fbSts7.rRobotAdjValue;
		ELSE
			PoseMirrorAdjustPrev := PoseMirrorAdjustPrevSts7;
			PoseMirrorAdjust := PoseMirrorAdjustPrevSts7;
			PoseMirrorAdjust[2] := PoseMirrorAdjustPrevSts7[2] - stStation.fbSts7.rRobotAdjValue;
		END_IF
	8: IF stStation.fbSts8.iAdjustmentCount < 1 THEN
			PoseMirrorAdjustPrev  := stStationPoses.aPoseMirrorPlaceSt3;
			PoseMirrorAdjust := stStationPoses.aPoseMirrorPlaceSt3;
			PoseMirrorAdjust[2] := stStationPoses.aPoseMirrorPlaceSt3[2] + stStation.fbSts8.rRobotAdjValue;
		ELSE
			PoseMirrorAdjustPrev := PoseMirrorAdjustPrevSts8;
			PoseMirrorAdjust := PoseMirrorAdjustPrevSts8;
			PoseMirrorAdjust[2] := PoseMirrorAdjustPrevSts8[2] - stStation.fbSts8.rRobotAdjValue;
		END_IF
	9: IF stStation.fbSts9.iAdjustmentCount < 1 THEN
			PoseMirrorAdjustPrev  := stStationPoses.aPoseMirrorPlaceSt3;
			PoseMirrorAdjust := stStationPoses.aPoseMirrorPlaceSt3;
			PoseMirrorAdjust[1] := stStationPoses.aPoseMirrorPlaceSt3[1] + stStation.fbSts9.rRobotAdjValue;
		ELSE
			PoseMirrorAdjustPrev := PoseMirrorAdjustPrevSts9;
			PoseMirrorAdjust := PoseMirrorAdjustPrevSts9;
			PoseMirrorAdjust[1] := PoseMirrorAdjustPrevSts9[1] - stStation.fbSts9.rRobotAdjValue;
		END_IF
	10: IF stStation.fbSts10.iAdjustmentCount < 1 THEN
			PoseMirrorAdjustPrev  := stStationPoses.aPoseMirrorPlaceSt3;
			PoseMirrorAdjust := stStationPoses.aPoseMirrorPlaceSt3;
			PoseMirrorAdjust[1] := stStationPoses.aPoseMirrorPlaceSt3[1] + stStation.fbSts10.rRobotAdjValue;
		ELSE
			PoseMirrorAdjustPrev := PoseMirrorAdjustPrevSts10;
			PoseMirrorAdjust := PoseMirrorAdjustPrevSts10;
			PoseMirrorAdjust[1] := PoseMirrorAdjustPrevSts10[1] - stStation.fbSts10.rRobotAdjValue;
		END_IF


END_CASE
END_METHOD

METHOD WritePoses : BOOL
VAR_INPUT
	iStationId : INT;
END_VAR
CASE iStationId OF // KORJAA POSE KIRJOTUS
	1: stStationPoses.aPoseLargeMotorPickupSt1 := stStation.stSts1.aPoseLargeMotorPickupSt1;
		stStationPoses.aPoseLargeMotorPickupSt2 := stStation.stSts1.aPoseLargeMotorPickupSt2;
		stStationPoses.aPoseLargeMotorPickupSt3 := stStation.stSts1.aPoseLargeMotorPickupSt3;
		stStationPoses.aPoseLargeMotorPlaceSt1 := stStation.stSts1.aPoseLargeMotorPlaceSt1;
		stStationPoses.aPoseLargeMotorPlaceSt2 := stStation.stSts1.aPoseLargeMotorPlaceSt2;
		stStationPoses.aPoseLargeMotorPlaceSt3 := stStation.stSts1.aPoseLargeMotorPlaceSt3;
		stStationPoses.aPoseMirrorAdj := stStation.stSts1.aPoseMirrorAdj;
		stStationPoses.aPoseMirrorPickupSt1 := stStation.stSts1.aPoseMirrorPickupSt1;
		stStationPoses.aPoseMirrorPickupSt2 := stStation.stSts1.aPoseMirrorPickupSt2;
		stStationPoses.aPoseMirrorPlaceSt1 := stStation.stSts1.aPoseG14MirrorPlaceSt1;
		stStationPoses.aPoseMirrorPlaceSt2 := stStation.stSts1.aPoseG14MirrorPlaceSt2;
		stStationPoses.aPoseMirrorPlaceSt3 := stStation.stSts1.aPoseG14MirrorPlaceSt3;
		stStationPoses.aPoseMirrorPlaceSt2[2] := stStation.stSts1.aPoseG14MirrorPlaceSt2[2] - rCouplerOffset - (15.05 - stAssemblyData.Station1To5.rMirrorGripPointOffsetToEdgeX + 1.2);
		stStationPoses.aPoseMirrorPlaceSt3[2] := stStation.stSts1.aPoseG14MirrorPlaceSt3[2] - rCouplerOffset - (15.05 - stAssemblyData.Station1To5.rMirrorGripPointOffsetToEdgeX + 0.7);
		stStationPoses.aPoseSmallMotorPlaceSt1 := stStation.stSts1.aPoseSmallMotorPlaceSt1;
		stStationPoses.aPoseSmallMotorPlaceSt2 := stStation.stSts1.aPoseSmallMotorPlaceSt2;
		stStationPoses.aPoseSmallMotorPickupSt1 := stStation.stSts1.aPoseSmallMotorPickupSt1;
		stStationPoses.aPoseSmallMotorPickupSt2 := stStation.stSts1.aPoseSmallMotorPickupSt2;
		stStationPoses.aPoseSmallMotorPickupSt3 := stStation.stSts1.aPoseSmallMotorPickupSt3;
		stStationPoses.aPosePassedLargeSt1 := stStation.stSts1.aPosePassedLargeSt1;
		stStationPoses.aPosePassedLargeSt2 := stStation.stSts1.aPosePassedLargeSt2;
		stStationPoses.aPosePassedLargeSt3 := stStation.stSts1.aPosePassedLargeSt3;
		stStationPoses.aPosePassedSmallSt1 := stStation.stSts1.aPosePassedSmallSt1;
		stStationPoses.aPosePassedSmallSt2 := stStation.stSts1.aPosePassedSmallSt2;
		stStationPoses.aPosePassedSmallSt3 := stStation.stSts1.aPosePassedSmallSt3;
		stStationPoses.rLinPosPalletPass := stStation.stSts1.rLinPosPalletPass;
		stStationPoses.rLinPosPalletReject := stStation.stSts1.rLinPosPalletReject;
		stStationPoses.rLinPosMotorPickup := stStation.stSts1.rLinPosMotorPickup;
		stStationPoses.rLinPosMirrorPickup := stStation.stSts1.rLinPosMirrorPickup;
		stStationPoses.rLinPosPlace := stStation.stSts1.rLinPosPlace;
		
	2: stStationPoses.aPoseLargeMotorPickupSt1 := stStation.stSts2.aPoseLargeMotorPickupSt1;
		stStationPoses.aPoseLargeMotorPickupSt2 := stStation.stSts2.aPoseLargeMotorPickupSt2;
		stStationPoses.aPoseLargeMotorPickupSt3 := stStation.stSts2.aPoseLargeMotorPickupSt3;
		stStationPoses.aPoseLargeMotorPlaceSt1 := stStation.stSts2.aPoseLargeMotorPlaceSt1;
		stStationPoses.aPoseLargeMotorPlaceSt2 := stStation.stSts2.aPoseLargeMotorPlaceSt2;
		stStationPoses.aPoseLargeMotorPlaceSt3 := stStation.stSts2.aPoseLargeMotorPlaceSt3;
		stStationPoses.aPoseMirrorAdj := stStation.stSts2.aPoseMirrorAdj;
		stStationPoses.aPoseMirrorPickupSt1 := stStation.stSts2.aPoseMirrorPickupSt1;
		stStationPoses.aPoseMirrorPickupSt2 := stStation.stSts2.aPoseMirrorPickupSt2;
		stStationPoses.aPoseMirrorPlaceSt1 := stStation.stSts2.aPoseG14MirrorPlaceSt1;
		stStationPoses.aPoseMirrorPlaceSt2 := stStation.stSts2.aPoseG14MirrorPlaceSt2;
		stStationPoses.aPoseMirrorPlaceSt3 := stStation.stSts2.aPoseG14MirrorPlaceSt3;
		stStationPoses.aPoseMirrorPlaceSt2[2] := stStation.stSts2.aPoseG14MirrorPlaceSt2[2] - rCouplerOffset - (15.05 - stAssemblyData.Station1To5.rMirrorGripPointOffsetToEdgeX + 1.2);
		stStationPoses.aPoseMirrorPlaceSt3[2] := stStation.stSts2.aPoseG14MirrorPlaceSt3[2] - rCouplerOffset - (15.05 - stAssemblyData.Station1To5.rMirrorGripPointOffsetToEdgeX + 0.7);
		stStationPoses.aPoseSmallMotorPlaceSt1 := stStation.stSts2.aPoseSmallMotorPlaceSt1;
		stStationPoses.aPoseSmallMotorPlaceSt2 := stStation.stSts2.aPoseSmallMotorPlaceSt2;
		stStationPoses.aPoseSmallMotorPickupSt1 := stStation.stSts2.aPoseSmallMotorPickupSt1;
		stStationPoses.aPoseSmallMotorPickupSt2 := stStation.stSts2.aPoseSmallMotorPickupSt2;
		stStationPoses.aPoseSmallMotorPickupSt3 := stStation.stSts2.aPoseSmallMotorPickupSt3;
		stStationPoses.aPosePassedLargeSt1 := stStation.stSts2.aPosePassedLargeSt1;
		stStationPoses.aPosePassedLargeSt2 := stStation.stSts2.aPosePassedLargeSt2;
		stStationPoses.aPosePassedLargeSt3 := stStation.stSts2.aPosePassedLargeSt3;
		stStationPoses.aPosePassedSmallSt1 := stStation.stSts2.aPosePassedSmallSt1;
		stStationPoses.aPosePassedSmallSt2 := stStation.stSts2.aPosePassedSmallSt2;
		stStationPoses.aPosePassedSmallSt3 := stStation.stSts2.aPosePassedSmallSt3;
		stStationPoses.aPosePassedSmallSt4 := stStation.stSts2.aPosePassedSmallSt4;
		stStationPoses.rLinPosPalletPass := stStation.stSts2.rLinPosPalletPass;
		stStationPoses.rLinPosPalletReject := stStation.stSts2.rLinPosPalletReject;
		stStationPoses.rLinPosMotorPickup := stStation.stSts2.rLinPosMotorPickup;
		stStationPoses.rLinPosMirrorPickup := stStation.stSts2.rLinPosMirrorPickup;
		stStationPoses.rLinPosPlace := stStation.stSts2.rLinPosPlace;
		
// 	3: stStationPoses.aPoseLargeMotorPickupSt1 := stStation.stSts3.aPoseLargeMotorPickupSt1;
// 		stStationPoses.aPoseLargeMotorPickupSt2 := stStation.stSts3.aPoseLargeMotorPickupSt2;
// 		stStationPoses.aPoseLargeMotorPickupSt3 := stStation.stSts3.aPoseLargeMotorPickupSt3;
// 		stStationPoses.aPoseLargeMotorPlaceSt1 := stStation.stSts3.aPoseLargeMotorPlaceSt1;
// 		stStationPoses.aPoseLargeMotorPlaceSt2 := stStation.stSts3.aPoseLargeMotorPlaceSt2;
// 		stStationPoses.aPoseLargeMotorPlaceSt3 := stStation.stSts3.aPoseLargeMotorPlaceSt3;
// 		stStationPoses.aPoseMirrorAdj := stStation.stSts3.aPoseMirrorAdj;
// 		stStationPoses.aPoseMirrorPickupSt1 := stStation.stSts3.aPoseMirrorPickupSt1;
// 		stStationPoses.aPoseMirrorPickupSt2 := stStation.stSts3.aPoseMirrorPickupSt2;
// 		stStationPoses.aPoseMirrorPlaceSt1 := stStation.stSts3.aPoseMirrorPlaceSt1;
// 		stStationPoses.aPoseMirrorPlaceSt2 := stStation.stSts3.aPoseMirrorPlaceSt2;
// 		stStationPoses.aPoseMirrorPlaceSt3 := stStation.stSts3.aPoseMirrorPlaceSt3;
// 		stStationPoses.aPoseSmallMotorPlaceSt1 := stStation.stSts3.aPoseSmallMotorPlaceSt1;
// 		stStationPoses.aPoseSmallMotorPlaceSt2 := stStation.stSts3.aPoseSmallMotorPlaceSt2;
// 		stStationPoses.aPoseSmallMotorPickupSt1 := stStation.stSts3.aPoseSmallMotorPickupSt1;
// 		stStationPoses.aPoseSmallMotorPickupSt2 := stStation.stSts3.aPoseSmallMotorPickupSt2;
// 		stStationPoses.aPoseSmallMotorPickupSt3 := stStation.stSts3.aPoseSmallMotorPickupSt3;
// 		stStationPoses.aPosePassedLargeSt1 := stStation.stSts3.aPosePassedLargeSt1;
// 		stStationPoses.aPosePassedLargeSt2 := stStation.stSts3.aPosePassedLargeSt2;
// 		stStationPoses.aPosePassedLargeSt3 := stStation.stSts3.aPosePassedLargeSt3;
// 		stStationPoses.aPosePassedSmallSt1 := stStation.stSts3.aPosePassedSmallSt1;
// 		stStationPoses.aPosePassedSmallSt2 := stStation.stSts3.aPosePassedSmallSt2;
// 		stStationPoses.aPosePassedSmallSt3 := stStation.stSts3.aPosePassedSmallSt3;
// 		stStationPoses.aPosePassedSmallSt4 := stStation.stSts3.aPosePassedSmallSt4;
// 		stStationPoses.rLinPosPalletPass := stStation.stSts3.rLinPosPalletPass;
// 		stStationPoses.rLinPosPalletReject := stStation.stSts3.rLinPosPalletReject;
// 		stStationPoses.rLinPosMotorPickup := stStation.stSts3.rLinPosMotorPickup;
// 		stStationPoses.rLinPosMirrorPickup := stStation.stSts3.rLinPosMirrorPickup;
// 		stStationPoses.rLinPosPlace := stStation.stSts3.rLinPosPlace;
END_CASE
END_METHOD

END_FUNCTION_BLOCK

// ---- POUs/Meca500/FB_linearAxisFunctions.TcPOU
FUNCTION_BLOCK FB_LinearAxisFunctions
VAR_INPUT
	stModuleHmi				: REFERENCE TO ST_ModuleHmi;
    stPlcCom                : REFERENCE TO ST_Module_PlcCom;
    ExecuteMovement         : BOOL;
    ExecuteHoming           : BOOL;
    AxisTargetPos           : LREAL;
    AxisVelo                : LREAL := 30;
    LinearHomingPosition    : LREAL := 0;
    AxisReset               : BOOL;
    bErrorClear             : BOOL;
END_VAR

VAR_OUTPUT
    bAxisStatusOK           : BOOL;
    CurrentPos              : LREAL;
    bError                  : BOOL;
    bMovementDone           : BOOL;
	bAxisHomed				: BOOL;
    ErrorID                 : UDINT;
    LinearAxisBusy          : BOOL;
END_VAR

VAR
    Axis1                   : AXIS_REF;
    fbPower1                : MC_Power;
    fbHome1                 : MC_Home;
    fbMoveAbs               : MC_MoveAbsolute;
    fbReset1                : MC_Reset;
    fbReadPos               : MC_ReadActualPosition;
    fbStatus                : MC_ReadStatus;
	fbJog					: MC_Jog;

    MasterState             : INT := 0;

    bAllowAbsMovement       : BOOL;
    bAbsMoveExecute         : BOOL;
    bHomeExec               : BOOL;
    bMoveExec               : BOOL;

    rHome                   : R_TRIG;
    rMove                   : R_TRIG;
    rReset                  : R_TRIG;
    rErrClear               : R_TRIG;

    MotionActive            : BOOL := FALSE;

    rAbsDone                : R_TRIG;
    tAbsDone                : TOF;
	stHomingOptions			: ST_HomingOptions;

    SafetyMain              : BOOL;
	bHomingJogState			: BOOL;
	iVelocity				: LREAL := 10;
END_VAR


////////////////////////////////////////////////////////////////////// Status reading
fbStatus(Axis := Axis1, Enable := TRUE);
fbReadPos(Axis := Axis1, Enable := TRUE);
CurrentPos := fbReadPos.Position;
SafetyMain := stPlcCom.stPlcComIn.bEstopOk AND stPlcCom.stPlcComIn.bSafetyOk;
bAxisStatusOK := fbStatus.Status.Operational AND NOT fbStatus.Error;


// Movement done tof
rAbsDone(CLK := fbMoveAbs.Done AND NOT fbMoveAbs.Error AND NOT fbMoveAbs.CommandAborted);
tAbsDone(IN := rAbsDone.Q, PT := T#500MS);
bMovementDone := tAbsDone.Q;


// Trigs
rHome(CLK := ExecuteHoming);
rMove(CLK := ExecuteMovement);
rReset(CLK := AxisReset);
stHomingOptions.SearchDirection := MC_Negative_Direction;
stHomingOptions.ClearPositionLag := TRUE;

// Movement execute
bAbsMoveExecute := bAllowAbsMovement AND rMove.Q;


// Busy
LinearAxisBusy := fbHome1.Busy OR fbMoveAbs.Busy OR fbReset1.Busy;

IF LinearAxisBusy THEN
    fbJog.JogForward := FALSE;
    fbJog.JogBackwards := FALSE;
END_IF


CASE MasterState OF

// Idle state
0:
    bError := FALSE;
    ErrorID := 0;
    bHomeExec := FALSE;
    bMoveExec := FALSE;
    bAbsMoveExecute := FALSE;
	bAxisHomed := FALSE;

    IF NOT stPlcCom.stPlcComIn.bSafetyOk THEN
        // Force movement disabled
        bAllowAbsMovement := FALSE;
        MasterState := 999;
	ELSIF NOT stPlcCom.stPlcComIn.bEstopOk THEN
		bAllowAbsMovement := FALSE;
		MasterState := 900;
    ELSIF NOT LinearAxisBusy THEN			// ELSIF rHome.Q AND NOT LinearAxisBusy THEN. // tämä rivi lisätty, kotiuttaa suoraan jos akseli vapaa ja safetyt ok
        MasterState := 10;
	END_IF
	
    IF rReset.Q THEN
        MasterState := 40;
    END_IF


// Power On

10:
    IF NOT stPlcCom.stPlcComIn.bSafetyOk THEN
        fbPower1.Enable := FALSE ;
        MasterState := 999;
	ELSIF NOT stPlcCom.stPlcComIn.bEstopOk THEN
		bAllowAbsMovement := FALSE;
		MasterState := 900;
    ELSE
        fbPower1.Enable := TRUE;
    END_IF

    IF fbPower1.Status THEN        
        MasterState := 15;		// was 20 before pre homing added

    ELSIF fbPower1.Error THEN
        bError := TRUE;
        ErrorID := fbPower1.ErrorID;
        MasterState := 1000;
    END_IF
	
	IF rReset.Q THEN
        MasterState := 40;
    END_IF
	
// Pre homing sensorCheck
15:
	IF NOT stPlcCom.stPlcComIn.bLinearAxisHomingSensor THEN		//Jog away from sensor if axis is on sensor at startup
		fbJog.JogForward := TRUE;
		bHomingJogState := TRUE;
	ELSE
		fbJog.JogForward := FALSE;						//Continue to regular homing once axis is off the sensor.
		IF fbJog.Done OR NOT bHomingJogState THEN
			bHomeExec := TRUE;
			bHomingJogState := FALSE;
			MasterState :=20;
		END_IF
	END_IF
	
	IF rReset.Q THEN
        MasterState := 40;
    END_IF
// Homing

20:
    IF NOT stPlcCom.stPlcComIn.bSafetyOk THEN
        bHomeExec := FALSE;
        MasterState := 999;
	ELSIF NOT stPlcCom.stPlcComIn.bEstopOk THEN
		bAllowAbsMovement := FALSE;
		MasterState := 900;
    END_IF

    IF fbHome1.Busy THEN
        MotionActive := TRUE;

    ELSIF fbHome1.Done OR fbHome1.CommandAborted OR fbHome1.Error THEN
        bHomeExec := FALSE;
        MotionActive := FALSE;

        IF fbHome1.Done THEN
            bAllowAbsMovement := TRUE;
            MasterState := 25;
			bAxisHomed := TRUE;
        ELSIF fbHome1.Error THEN
            bError := TRUE;
            ErrorID := fbHome1.ErrorID;
            MasterState := 1000;
        ELSE
            MasterState := 0;
        END_IF
    END_IF

    IF rReset.Q THEN
        bHomeExec := FALSE;
        MasterState := 40;
    END_IF


//  Idle after homing

25:
    IF fbPower1.Error OR fbHome1.Error OR fbMoveAbs.Error OR fbReset1.Error THEN
        bError := TRUE;

        IF fbMoveAbs.Error THEN ErrorID := fbMoveAbs.ErrorID;
        ELSIF fbHome1.Error THEN ErrorID := fbHome1.ErrorID;
        ELSIF fbPower1.Error THEN ErrorID := fbPower1.ErrorID;
        ELSIF fbReset1.Error THEN ErrorID := fbReset1.ErrorID;
        END_IF

        MasterState := 1000;

    ELSIF bAbsMoveExecute AND stPlcCom.stPlcComIn.bEstopOk AND stPlcCom.stPlcComIn.bSafetyOk AND NOT LinearAxisBusy AND AxisTargetPos < 420.1 THEN
        bMoveExec := TRUE;
        bMovementDone := FALSE;
        MasterState := 30;

    ELSIF NOT stPlcCom.stPlcComIn.bSafetyOk THEN
        bAllowAbsMovement := FALSE;
        MasterState := 999;
		
	ELSIF NOT stPlcCom.stPlcComIn.bEstopOk THEN
		bAllowAbsMovement := FALSE;
		MasterState := 900;
    END_IF
	IF CurrentPos < 0.1 AND CurrentPos > -0.1 THEN
		bAxisHomed := TRUE;
	ELSE
		bAxisHomed := FALSE;
	END_IF
	
	IF stModuleHmi.MecaHmi.bLinearJogScreenActive AND stPlcCom.stPlcComIn.bSafetyOk AND stPlcCom.stPlcComIn.bEstopOk AND NOT LinearAxisBusy AND NOT AxisReset THEN
	MasterState := 100;
	ELSIF NOT stModuleHmi.MecaHmi.bLinearJogScreenActive THEN
    	fbJog.JogForward := FALSE;
    	fbJog.JogBackwards := FALSE;
	ELSIF rReset.Q THEN
		MasterState :=40;   
	END_IF
	
	IF rReset.Q THEN
		MasterState := 40;
	END_IF
// Absolute Move

30:
    IF NOT stPlcCom.stPlcComIn.bSafetyOk THEN
        bMoveExec := FALSE;
        MasterState := 999;
		
	ELSIF NOT stPlcCom.stPlcComIn.bEstopOk THEN
		bAllowAbsMovement := FALSE;
		MasterState := 900;
    END_IF
	
    IF fbMoveAbs.Busy THEN
        MotionActive := TRUE;

    ELSIF fbMoveAbs.Done OR fbMoveAbs.CommandAborted OR fbMoveAbs.Error THEN
        bMoveExec := FALSE;
        MotionActive := FALSE;

        IF fbMoveAbs.Done THEN
            MasterState := 25;

        ELSIF fbMoveAbs.Error THEN
            bError := TRUE;
            ErrorID := fbMoveAbs.ErrorID;
            MasterState := 1000;
        ELSE
            MasterState := 25;
        END_IF
    END_IF

    IF rReset.Q THEN
        bMoveExec := FALSE;
        MasterState := 40;
    END_IF


// Reset sequence

40:
    fbReset1.Execute := TRUE;

    IF fbReset1.Done THEN
        fbReset1.Execute := FALSE;
        bAllowAbsMovement := FALSE;
        fbPower1.Enable := FALSE;
        MasterState := 0;

    ELSIF fbReset1.Error THEN
        bError := TRUE;
        ErrorID := fbReset1.ErrorID;
        MasterState := 1000;
    END_IF

100: // Manual movements
		IF fbMoveAbs.Done THEN
			bMoveExec := FALSE;
		END_IF
		AxisTargetPos := stModuleHmi.MecaHmi.rManualTargetPos;
		
		IF stModuleHmi.MecaHmi.bLinearJogScreenActive THEN
			IF stModuleHmi.MecaHmi.bJogLinearPositive AND NOT stModuleHmi.MecaHmi.bJogLinearNegative THEN
			    IF CurrentPos < 410 THEN
			        IF iVelocity <> 10 THEN
			            fbJog.JogForward := FALSE;
			            iVelocity := 10;
			        ELSE
			            fbJog.JogForward := TRUE;
			        END_IF
			    ELSIF CurrentPos < 420 THEN
			        IF iVelocity <> 3 THEN
			            fbJog.JogForward := FALSE;
			            iVelocity := 3;
			        ELSE
			            fbJog.JogForward := TRUE;
			        END_IF
			    END_IF
			ELSIF NOT stModuleHmi.MecaHmi.bJogLinearPositive THEN
			    fbJog.JogForward := FALSE;
			END_IF

			IF stModuleHmi.MecaHmi.bJogLinearNegative AND NOT stModuleHmi.MecaHmi.bJogLinearPositive THEN
			    IF CurrentPos > 10 THEN
			        IF iVelocity <> 10 THEN
			            fbJog.JogBackwards := FALSE;
			            iVelocity := 10;
			        ELSE
			            fbJog.JogBackwards := TRUE;
			        END_IF
			    ELSIF CurrentPos > 4 THEN
			        IF iVelocity <> 3 THEN
			            fbJog.JogBackwards := FALSE;
			            iVelocity := 3;
			        ELSE
			            fbJog.JogBackwards := TRUE;
			        END_IF
			    END_IF
			ELSIF NOT stModuleHmi.MecaHmi.bJogLinearNegative THEN
			    fbJog.JogBackwards := FALSE;
			END_IF
			
			IF fbMoveAbs.Error OR fbMoveAbs.CommandAborted THEN
    				bError := TRUE;
    				ErrorID := fbMoveAbs.ErrorID;
    				MasterState := 1000;
				ELSIF stModuleHmi.MecaHmi.bManualAbsMove AND stPlcCom.stPlcComIn.bEstopOk AND stPlcCom.stPlcComIn.bSafetyOk AND NOT LinearAxisBusy AND AxisTargetPos < 420.1 AND AxisTargetPos > 0.0 THEN
					bMoveExec := TRUE;
			END_IF
    		
			IF fbMoveAbs.Done AND stModuleHmi.MecaHmi.bManualAbsMove THEN
				stModuleHmi.MecaHmi.bManualAbsMove := FALSE;
			END_IF
			
			IF rReset.Q THEN
        		bMoveExec := FALSE;
        		MasterState := 40;
    		END_IF
	
		ELSE
			MasterState := 25;
		END_IF
		
		IF rReset.Q THEN
        		bMoveExec := FALSE;
        		MasterState := 40;
    		END_IF
		
900:
    bError := TRUE;
    ErrorID := 900;

    bHomeExec := FALSE;
    bMoveExec := FALSE;
    bAbsMoveExecute := FALSE;
    bAllowAbsMovement := FALSE;			//See if this works

    IF stPlcCom.stPlcComIn.bEstopOk AND rHome.Q THEN	  // Safety OK, go to reset
        MasterState := 0;
    END_IF
	
	IF stPlcCom.stPlcComIn.bEstopOk AND rReset.Q THEN
		MasterState := 40;
	END_IF

// Safety Fault 
999:
    ErrorID := 999;
	bAxisHomed := FALSE;
    bHomeExec := FALSE;
    bMoveExec := FALSE;
    bAbsMoveExecute := FALSE;
    bAllowAbsMovement := FALSE;

    IF stPlcCom.stPlcComIn.bSafetyOk AND rHome.Q THEN  // Safety OK, go to reset
        MasterState := 0;
    END_IF
	
	IF stPlcCom.stPlcComIn.bSafetyOk AND rReset.Q THEN
		MasterState := 40;
	END_IF

// Error state

1000:
    bError := TRUE;
    bHomeExec := FALSE;
    bMoveExec := FALSE;
	bAxisHomed := FALSE;
    IF rReset.Q THEN
        MasterState := 40;
    END_IF


END_CASE


fbJog(Axis:=Axis1, Velocity:=iVelocity, Acceleration :=458.796, Deceleration:=458.796,Jerk:=1376.388, Mode:=E_JogMode.MC_JOGMODE_CONTINOUS);

fbHome1(
	Axis            := Axis1,
	Execute         := bHomeExec,
	Position        := LinearHomingPosition,
	Options 		:= stHomingOptions,
	bCalibrationCam := stPlcCom.stPlcComIn.bLinearAxisHomingSensor );

fbPower1(
	Axis := Axis1,
	Enable_Positive := TRUE,
	Enable_Negative := TRUE);
	
fbReset1(Axis := Axis1);

fbMoveAbs(
	Axis         := Axis1,
	Execute      := bMoveExec,
	Position     := AxisTargetPos,
	Velocity     := AxisVelo,
	Acceleration := 0,
	Deceleration := 0,
	BufferMode   := MC_BufferMode.MC_Aborting);

END_FUNCTION_BLOCK

// ---- POUs/Meca500/Op/FB_GluingTipPositioning.TcPOU
FUNCTION_BLOCK FB_GluingTipPositioning
VAR_INPUT
	bExecutePositining : BOOL;
	stPlcCom	: REFERENCE TO ST_Module_PlcCom;
	rJogSpeed : REFERENCE TO REAL;
	bReCheckNeedle : BOOL;
END_VAR
VAR_OUTPUT
	bRobotHomed : BOOL;
	bDetectionDone : BOOL;
	bReDetectionDone : BOOL;
	bDetectionFailed	: BOOL;
	stTipOffsets	: ST_GluetipCoordinates;
END_VAR
VAR
	Sent				: BOOL;
	Buffered			: BOOL;
	Error				: BOOL;
	
	Delay				:Meca500_Delay;
	Gripper				:Meca500_Gripper;
	MoveGripper			:Meca500_MoveGripper;
	MoveJoints			:Meca500_MoveJoints;
	MoveJointsRel		:Meca500_MoveJointsRel;
	MovejointsVel		:Meca500_MoveJointsVel;
	MoveLin				:Meca500_MoveLin;
	MoveLinRelTrf		:Meca500_MoveLinRelTrf;
	MoveLinRelWrf		:Meca500_MoveLinRelWrf;
	MoveLinVelTrf		:Meca500_MoveLinVelTrf;
	MoveLinVelWrf		:Meca500_MoveLinVelWrf;
	MovePose			:Meca500_MovePose;
	SetAutoConf			:Meca500_SetAutoConf;
	SetAutoConfTurn		:Meca500_SetAutoConfTurn;
	SetBlending			:Meca500_SetBlending;
	SetCartAcc			:Meca500_SetCartAcc;
	SetCartAngVel		:Meca500_SetCartAngVel;
	SetCartLinVel		:Meca500_SetCartLinVel;
	SetCheckpoint		:Meca500_SetCheckpoint;
	SetConf				:Meca500_SetConf;
	SetConfTurn			:Meca500_SetConfTurn;
	SetGripperForce		:Meca500_SetGripperForce;
	SetGripperRange		:Meca500_SetGripperRange;
	SetGripperVel		:Meca500_SetGripperVel;
	SetJointAcc			:Meca500_SetJointAcc;
	SetJointVel			:Meca500_SetJointVel;
	SetTorqueLimitCfg	:Meca500_SetTorqueLimitCfg;
	SetTorqueLimits		:Meca500_SetTorqueLimits;
	SetTrf				:Meca500_SetTrf;
	SetValveState		:Meca500_SetValveState;
	SetVelTimeout		:Meca500_SetVelTimeout;
	SetWrf				:Meca500_SetWrf;
	StartProgram		:Meca500_StartProgram;
	SetJointVelLimit	:Meca500_SetJointVelLimit;
	SetTimeScaling		:Meca500_SetTimeScaling;
	GetEOAT 			:Meca500_GetEOAT;
	
	
	
	iPositioningStep	: INT;
	
	aNegativeJogZ				: ARRAY [1..6] OF REAL := [0,0,-0.2,0,0,0];
	
	PoseHome			: ARRAY [1..6] OF REAL := [-90,0,0,0,90,0];
	PoseMotorPickupTemp : ARRAY [1..6] OF REAL := [-73.2067 , 21.8881 , 23.8300 , -105.4797 , 75.4102 , -42.2884]; // JOINT VALUES
	PoseMotorPlaceTemp 	: ARRAY [1..6] OF REAL := [127.3581 , -0.6526 , 7.9110 , 0.0000 , 82.7417, 37.3370]; // JOINT VALUES
	PoseMirrorPickupTemp : ARRAY [1..6] OF REAL := [-154.1223 , 13.9826 , 1.7675 , 0.0000 ,  74.2499, 27.9110]; // JOINT VALUES
	PoseMidPose 		: ARRAY [1..6] OF REAL := [-150.872, 152.243,154.566, -119.571, -22.210 ,84.857]; // 
	
	PoseTipSt1		:  ARRAY [1..6] OF REAL := [-179.478, 170.365 , 101.774  , -119.571 , -22.210 , 84.857]; // Mid station before detection 1
	PoseTipSt2 		:  ARRAY [1..6] OF REAL := [-206.937, 217.033 , 86.60 , -100, -10 ,90]; // Pose start of detection 1
	PoseTipSt3 		:  ARRAY [1..6] OF REAL := [-207.937, 222.033 ,86.60 , -100, -10 ,90]; // Pose end of detection 1 92.875
	
	PoseTipSt4		:  ARRAY [1..6] OF REAL := [-170.757, 186.867 ,163.452 , -100, -40 ,90]; // Mid pose after first detection
	PoseTipSt5 		:  ARRAY [1..6] OF REAL := [-198.342, 212.81,92.875 , -115, -38 ,75.268]; // Pose start of detection 2
	PoseTipSt6 		:  ARRAY [1..6] OF REAL := [-202.667, 218.711,92.875 , -115, -38 ,75.268]; // Pose end of detection 2
	PoseTipFound 		:  ARRAY [1..6] OF REAL := [-198.937, 225.033 ,85.875 , -100, -10 ,90];
	PoseTipFoundEnd	:  ARRAY [1..6] OF REAL := [-198.937, 225.033 ,85.875 , -100, -10 ,90];
	EOAT				: ARRAY [0..5] OF REAL; // Values: [holding part, desired fingers opening reached, gripper closed, gripper open, gripper force, fingers opening].
	
	bMoveForward	: BOOL;
	rDetectedTipPosY : REAL;
	rDetectedTipPosX : REAL;
	bSaveFirstCoordinates : BOOL;
	bSaveSecondCoordinates : BOOL;
	bSaveThirdCoordinates : BOOL;
	aDetectedCoordinates	: ARRAY [1..4] OF ST_GluetipCoordinates;
	rSetpointX				: REAL := -201.8805;
	rSetPointY				: REAL := 219.1602;
	rSetPointZ				: REAL := 87.286;
	iSavingNumber	: INT;
	CoordinateSaveTrig	: R_TRIG;
	bNeedleFound : BOOL;
	bTrigPositionSave: BOOL;
	bHolt : BOOL;
	bHeightSet: BOOL;
	bPositionSaved: BOOL;
	bPassStepSent : BOOL;
	bMoveDown : BOOL;
	bNeedleDetected :BOOL;
	bAllowReCheck : BOOL;
END_VAR

GetEOAT(
	Status => EOAT,
	Robot := Meca500.GVL.Meca500);
IF NOT stPlcCom.stPlcComIn.bRobotGripperSensor THEN
	bNeedleFound := TRUE;
END_IF

bDetectionDone := FALSE;
bReDetectionDone := FALSE;
CoordinateSaveTrig(CLK := bNeedleFound);
IF CoordinateSaveTrig.Q AND bSaveFirstCoordinates THEN
	aDetectedCoordinates[1].X := Meca500.GVL.Meca500.Inputs.End_Effector_Pose.SubIndex_001;
	aDetectedCoordinates[1].Y := Meca500.GVL.Meca500.Inputs.End_Effector_Pose.SubIndex_002;
	aDetectedCoordinates[1].Z := Meca500.GVL.Meca500.Inputs.End_Effector_Pose.SubIndex_003;
	bSaveFirstCoordinates := FALSE;
END_IF

IF bSaveSecondCoordinates THEN
	aDetectedCoordinates[2].X := Meca500.GVL.Meca500.Inputs.End_Effector_Pose.SubIndex_001;
	aDetectedCoordinates[2].Y := Meca500.GVL.Meca500.Inputs.End_Effector_Pose.SubIndex_002;
	aDetectedCoordinates[2].Z := Meca500.GVL.Meca500.Inputs.End_Effector_Pose.SubIndex_003;
	bSaveSecondCoordinates := FALSE;
END_IF

IF CoordinateSaveTrig.Q AND bSaveThirdCoordinates THEN
	aDetectedCoordinates[3].X := Meca500.GVL.Meca500.Inputs.End_Effector_Pose.SubIndex_001;
	aDetectedCoordinates[3].Y := Meca500.GVL.Meca500.Inputs.End_Effector_Pose.SubIndex_002;
	aDetectedCoordinates[3].Z := Meca500.GVL.Meca500.Inputs.End_Effector_Pose.SubIndex_003;
	bSaveThirdCoordinates := FALSE;
END_IF
IF NOT stPlcCom.stPlcComIn.bRobotGripperSensor AND bAllowReCheck THEN
	bNeedleDetected := TRUE;
	bAllowReCheck := FALSE;
END_IF

CASE iPositioningStep OF
	0: IF bExecutePositining AND NOT bReCheckNeedle THEN
			bDetectionDone := FALSE;
			bRobotHomed := FALSE;
			bNeedleFound := FALSE;
			bNeedleDetected := FALSE;
			bReDetectionDone := FALSE;
			bDetectionFailed := FALSE;			
			PoseTipSt2[3] := 86.6;
			PoseTipSt3[3] := 86.6;			
			IF NOT stPlcCom.stPlcComIn.bGlueStopHome THEN
				iPositioningStep := 1;
				bExecutePositining := FALSE;
			ELSE
				stPlcCom.stPlcComOut.bGlueStopValve := TRUE;
			END_IF
		ELSIF bExecutePositining AND bReCheckNeedle THEN
			iPositioningStep := 50;
			bExecutePositining := FALSE;
			bReCheckNeedle := FALSE;
		END_IF
	1: MoveGripper(mm := 24,
			ExternalStatecontrol := 0,
			ExternalMove_ID := 0,
			Robot:= Meca500.GVL.Meca500, 
			Error=> Error, 
			Sent:= Sent, 
			Buffered:= Buffered);
	2:	IF EOAT[5] = 24 THEN  // LISÄÄ ELSE
			iPositioningStep := 3;
		END_IF
	3: MoveJoints(Joint_Angle := PoseMotorPlaceTemp,
			ExternalStatecontrol := 0,
			ExternalMove_ID := 0,
			Robot:= Meca500.GVL.Meca500, 
			Error=> Error, 
			Sent:= Sent, 
			Buffered:= Buffered);
	4: MovePose(Pose := PoseMidPose,
			ExternalStatecontrol := 0,
			ExternalMove_ID := 0,
			Robot:= Meca500.GVL.Meca500, 
			Error=> Error, 
			Sent:= Sent, 
			Buffered:= Buffered);
	5: SetCheckpoint(CheckpointID := 201,
			ExternalStatecontrol := 0,
			ExternalMove_ID := 0,
			Robot:= Meca500.GVL.Meca500, 
			Error=> Error, 
			Sent:= Sent, 
			Buffered:= Buffered);
	6:	IF Meca500.GVL.Meca500.Inputs.Motion_Status.ReachedCheckPointId = 201 THEN
			iPositioningStep := 7;	
		END_IF
	 
	7: MovePose(Pose := PoseTipSt1,
			ExternalStatecontrol := 0,
			ExternalMove_ID := 0,
			Robot:= Meca500.GVL.Meca500, 
			Error=> Error, 
			Sent:= Sent, 
			Buffered:= Buffered);	
	8: SetCheckpoint(CheckpointID := 203,
			ExternalStatecontrol := 0,
			ExternalMove_ID := 0,
			Robot:= Meca500.GVL.Meca500, 
			Error=> Error, 
			Sent:= Sent, 
			Buffered:= Buffered);
	9: IF Meca500.GVL.Meca500.Inputs.Motion_Status.ReachedCheckPointId = 203 THEN
			bHeightSet := FALSE;
			bSaveFirstCoordinates := TRUE;
			iPositioningStep := 10;
		END_IF 
	10: MoveLin(Pose := PoseTipSt2,
			ExternalStatecontrol := 0,
			ExternalMove_ID := 0,
			Robot:= Meca500.GVL.Meca500, 
			Error=> Error, 
			Sent:= Sent, 
			Buffered:= Buffered);
	11: SetCartLinVel(
			Velocity_Limit := 0.25,
			ExternalStatecontrol := 0,
			ExternalMove_ID := 0,
			Robot:= Meca500.GVL.Meca500, 
			Error=> Error, 
			Sent:= Sent, 
			Buffered:= Buffered);
	12: MoveLin(Pose := PoseTipSt3,
			ExternalStatecontrol := 0,
			ExternalMove_ID := 0,
			Robot:= Meca500.GVL.Meca500, 
			Error=> Error, 
			Sent:= Sent, 
			Buffered:= Buffered);
	
	13: SetCheckpoint(CheckpointID := 202,
			ExternalStatecontrol := 0,
			ExternalMove_ID := 0,
			Robot:= Meca500.GVL.Meca500, 
			Error=> Error, 
			Sent:= Sent, 
			Buffered:= Buffered);
	14:	IF Meca500.GVL.Meca500.Inputs.Motion_Status.ReachedCheckPointId = 202 THEN
			IF bNeedleFound THEN
				iPositioningStep := 15;	
			ELSIF PoseTipSt2[3] < 94 AND NOT bHeightSet THEN
				PoseTipSt2[3] := PoseTipSt2[3] + 0.5;
				PoseTipSt3[3] := PoseTipSt3[3] + 0.5;
				bHeightSet := TRUE;
				iPositioningStep := 8;	
			ELSE
				iPositioningStep := 100; 
			END_IF
		END_IF	
	15: SetCartLinVel(
			Velocity_Limit := 10*rJogSpeed,
			ExternalStatecontrol := 0,
			ExternalMove_ID := 0,
			Robot:= Meca500.GVL.Meca500, 
			Error=> Error, 
			Sent:= Sent, 
			Buffered:= Buffered);
	16: PoseTipFound[1] := aDetectedCoordinates[1].X;
		PoseTipFound[2] := aDetectedCoordinates[1].Y;
		PoseTipFound[3] := aDetectedCoordinates[1].Z;
		bNeedleFound := FALSE;
		iPositioningStep := 17;
	17: MovePose(Pose := PoseTipFound, // LISÄÄ KOODI JOSSA JOS PALUU POSITIOON EI OLE NEULAN KOHDALLA NIIN TUNNISTUS ALKAA ALUSTA
			ExternalStatecontrol := 0,
			ExternalMove_ID := 0,
			Robot:= Meca500.GVL.Meca500, 
			Error=> Error, 
			Sent:= Sent, 
			Buffered:= Buffered);
	18: SetCheckpoint(CheckpointID := 205,
			ExternalStatecontrol := 0,
			ExternalMove_ID := 0,
			Robot:= Meca500.GVL.Meca500, 
			Error=> Error, 
			Sent:= Sent, 
			Buffered:= Buffered);
			
	19: IF Meca500.GVL.Meca500.Inputs.Motion_Status.ReachedCheckPointId = 205 THEN
			iPositioningStep := 20;
			PoseTipSt1[3] := 92;
		END_IF
		
	20: bPassStepSent := TRUE;
		IF bMoveDown THEN
			 MoveLinVelWrf(
				Velocity := aNegativeJogZ,
				ExternalStatecontrol := 0,
				ExternalMove_ID := 0,
				Robot:= Meca500.GVL.Meca500, 
				Error=> Error, 
				Sent:= Sent, 
				Buffered:= Buffered);
		END_IF
		IF Meca500.GVL.Meca500.Inputs.End_Effector_Pose.SubIndex_003 < 81 THEN
			iPositioningStep := 100; 
			bMoveDown := FALSE;
		ELSIF NOT stPlcCom.stPlcComIn.bRobotGripperSensor THEN
			bMoveDown := TRUE;
		ELSE
			bSaveSecondCoordinates := TRUE;
			bMoveDown := FALSE;
			iPositioningStep := 21;
			bPassStepSent := FALSE;
		END_IF
		IF Sent AND Buffered THEN
			Sent := FALSE;
			Buffered := FALSE;
		END_IF	
		
	21: MoveLin(Pose := PoseTipSt2,
			ExternalStatecontrol := 0,
			ExternalMove_ID := 0,
			Robot:= Meca500.GVL.Meca500, 
			Error=> Error, 
			Sent:= Sent, 
			Buffered:= Buffered);
	22: MoveLin(Pose := PoseTipSt1,
			ExternalStatecontrol := 0,
			ExternalMove_ID := 0,
			Robot:= Meca500.GVL.Meca500, 
			Error=> Error, 
			Sent:= Sent, 
			Buffered:= Buffered);
	23: MovePose(Pose := PoseMidPose,
			ExternalStatecontrol := 0,
			ExternalMove_ID := 0,
			Robot:= Meca500.GVL.Meca500, 
			Error=> Error, 
			Sent:= Sent, 
			Buffered:= Buffered);	
	24: MoveJoints(Joint_Angle := PoseMotorPlaceTemp,
			ExternalStatecontrol := 0,
			ExternalMove_ID := 0,
			Robot:= Meca500.GVL.Meca500, 
			Error=> Error, 
			Sent:= Sent, 
			Buffered:= Buffered);
	25:	SetCheckpoint(CheckpointID := 207,
			ExternalStatecontrol := 0,
			ExternalMove_ID := 0,
			Robot:= Meca500.GVL.Meca500, 
			Error=> Error, 
			Sent:= Sent, 
			Buffered:= Buffered);
	26: IF Meca500.GVL.Meca500.Inputs.Motion_Status.ReachedCheckPointId = 207 THEN
			iPositioningStep := 27;
			bNeedleFound := FALSE;
			PoseTipSt5[3] := aDetectedCoordinates[1].Z + 1;
			PoseTipSt6[3] := aDetectedCoordinates[1].Z + 1;
		END_IF
	27: MovePose(Pose := PoseTipSt4,
			ExternalStatecontrol := 0,
			ExternalMove_ID := 0,
			Robot:= Meca500.GVL.Meca500, 
			Error=> Error, 
			Sent:= Sent, 
			Buffered:= Buffered);
	28: MovePose(Pose := PoseTipSt5,
			ExternalStatecontrol := 0,
			ExternalMove_ID := 0,
			Robot:= Meca500.GVL.Meca500, 
			Error=> Error, 
			Sent:= Sent, 
			Buffered:= Buffered);
	29: SetCartLinVel(
			Velocity_Limit := 0.25,
			ExternalStatecontrol := 0,
			ExternalMove_ID := 0,
			Robot:= Meca500.GVL.Meca500, 
			Error=> Error, 
			Sent:= Sent, 
			Buffered:= Buffered);
	30: SetCheckpoint(CheckpointID := 208,
			ExternalStatecontrol := 0,
			ExternalMove_ID := 0,
			Robot:= Meca500.GVL.Meca500, 
			Error=> Error, 
			Sent:= Sent, 
			Buffered:= Buffered);
	31: IF Meca500.GVL.Meca500.Inputs.Motion_Status.ReachedCheckPointId = 208 THEN
			iPositioningStep := 32;
			bSaveThirdCoordinates := TRUE;
			bHeightSet := FALSE;
		END_IF
	32: MoveLin(Pose := PoseTipSt6,
			ExternalStatecontrol := 0,
			ExternalMove_ID := 0,
			Robot:= Meca500.GVL.Meca500, 
			Error=> Error, 
			Sent:= Sent, 
			Buffered:= Buffered);
	33: SetCartLinVel(
			Velocity_Limit := 10*rJogSpeed,
			ExternalStatecontrol := 0,
			ExternalMove_ID := 0,
			Robot:= Meca500.GVL.Meca500, 
			Error=> Error, 
			Sent:= Sent, 
			Buffered:= Buffered);
	34: MovePose(Pose := PoseTipSt5,
			ExternalStatecontrol := 0,
			ExternalMove_ID := 0,
			Robot:= Meca500.GVL.Meca500, 
			Error=> Error, 
			Sent:= Sent, 
			Buffered:= Buffered);
	35: MovePose(Pose := PoseTipSt4,
			ExternalStatecontrol := 0,
			ExternalMove_ID := 0,
			Robot:= Meca500.GVL.Meca500, 
			Error=> Error, 
			Sent:= Sent, 
			Buffered:= Buffered);
	36: MoveJoints(Joint_Angle := PoseMotorPlaceTemp,
			ExternalStatecontrol := 0,
			ExternalMove_ID := 0,
			Robot:= Meca500.GVL.Meca500, 
			Error=> Error, 
			Sent:= Sent, 
			Buffered:= Buffered);
	37: SetCheckpoint(CheckpointID := 209,
			ExternalStatecontrol := 0,
			ExternalMove_ID := 0,
			Robot:= Meca500.GVL.Meca500, 
			Error=> Error, 
			Sent:= Sent, 
			Buffered:= Buffered);
	38: IF Meca500.GVL.Meca500.Inputs.Motion_Status.ReachedCheckPointId = 209 THEN
			stPlcCom.stPlcComOut.bGlueStopValve := FALSE;
			stTipOffsets.X := rSetpointX- aDetectedCoordinates[3].X;
			stTipOffsets.Y := rSetpointY- aDetectedCoordinates[2].Y;
			stTipOffsets.Z := rSetpointZ- aDetectedCoordinates[2].Z;
			iPositioningStep := 39;
		END_IF
	39: bDetectionDone := TRUE;
		iPositioningStep := 0;
	50:MoveGripper(mm := 24,
			ExternalStatecontrol := 0,
			ExternalMove_ID := 0,
			Robot:= Meca500.GVL.Meca500, 
			Error=> Error, 
			Sent:= Sent, 
			Buffered:= Buffered);
	51:	IF EOAT[5] = 24 THEN  // LISÄÄ ELSE
			PoseTipFound[3] := PoseTipFound[3]+1;
			PoseTipFoundEnd := PoseTipFound;
			PoseTipFound[2] := PoseTipFound[2] - 0.3;
			PoseTipFoundEnd[2] :=  PoseTipFoundEnd[2]+ 0.3;
			bAllowReCheck := TRUE;
			iPositioningStep := 52;
		END_IF
	52: MoveJoints(Joint_Angle := PoseMotorPlaceTemp,
			ExternalStatecontrol := 0,
			ExternalMove_ID := 0,
			Robot:= Meca500.GVL.Meca500, 
			Error=> Error, 
			Sent:= Sent, 
			Buffered:= Buffered);
	53: MovePose(Pose := PoseMidPose,
			ExternalStatecontrol := 0,
			ExternalMove_ID := 0,
			Robot:= Meca500.GVL.Meca500, 
			Error=> Error, 
			Sent:= Sent, 
			Buffered:= Buffered);
	54: SetCheckpoint(CheckpointID := 201,
			ExternalStatecontrol := 0,
			ExternalMove_ID := 0,
			Robot:= Meca500.GVL.Meca500, 
			Error=> Error, 
			Sent:= Sent, 
			Buffered:= Buffered);
	55:	IF Meca500.GVL.Meca500.Inputs.Motion_Status.ReachedCheckPointId = 201 THEN
			iPositioningStep := 56;	
		END_IF
	 
	56: MovePose(Pose := PoseTipSt1,
			ExternalStatecontrol := 0,
			ExternalMove_ID := 0,
			Robot:= Meca500.GVL.Meca500, 
			Error=> Error, 
			Sent:= Sent, 
			Buffered:= Buffered);	
	57: SetCheckpoint(CheckpointID := 203,
			ExternalStatecontrol := 0,
			ExternalMove_ID := 0,
			Robot:= Meca500.GVL.Meca500, 
			Error=> Error, 
			Sent:= Sent, 
			Buffered:= Buffered);
	58: IF Meca500.GVL.Meca500.Inputs.Motion_Status.ReachedCheckPointId = 203 THEN
			bHeightSet := FALSE;
			bSaveFirstCoordinates := TRUE;
			iPositioningStep := 59;
			stPlcCom.stPlcComOut.bGlueStopValve := TRUE;
		END_IF 
	59: MoveLin(Pose := PoseTipSt2,
			ExternalStatecontrol := 0,
			ExternalMove_ID := 0,
			Robot:= Meca500.GVL.Meca500, 
			Error=> Error, 
			Sent:= Sent, 
			Buffered:= Buffered);
	60: MoveLin(Pose := PoseTipFound,
			ExternalStatecontrol := 0,
			ExternalMove_ID := 0,
			Robot:= Meca500.GVL.Meca500, 
			Error=> Error, 
			Sent:= Sent, 
			Buffered:= Buffered); 
	61: SetCartLinVel(
			Velocity_Limit := 0.25,
			ExternalStatecontrol := 0,
			ExternalMove_ID := 0,
			Robot:= Meca500.GVL.Meca500, 
			Error=> Error, 
			Sent:= Sent, 
			Buffered:= Buffered);
	62: SetCheckpoint(CheckpointID := 203,
			ExternalStatecontrol := 0,
			ExternalMove_ID := 0,
			Robot:= Meca500.GVL.Meca500, 
			Error=> Error, 
			Sent:= Sent, 
			Buffered:= Buffered);
	63: IF Meca500.GVL.Meca500.Inputs.Motion_Status.ReachedCheckPointId = 203 THEN
			iPositioningStep := 64;
		END_IF
	64: MoveLin(Pose := PoseTipFoundEnd,
			ExternalStatecontrol := 0,
			ExternalMove_ID := 0,
			Robot:= Meca500.GVL.Meca500, 
			Error=> Error, 
			Sent:= Sent, 
			Buffered:= Buffered);
	65: SetCheckpoint(CheckpointID := 200,
			ExternalStatecontrol := 0,
			ExternalMove_ID := 0,
			Robot:= Meca500.GVL.Meca500, 
			Error=> Error, 
			Sent:= Sent, 
			Buffered:= Buffered);
	66: IF Meca500.GVL.Meca500.Inputs.Motion_Status.ReachedCheckPointId = 200 THEN
			iPositioningStep := 67;
		END_IF
	67: SetCartLinVel(
			Velocity_Limit := 10*rJogSpeed,
			ExternalStatecontrol := 0,
			ExternalMove_ID := 0,
			Robot:= Meca500.GVL.Meca500, 
			Error=> Error, 
			Sent:= Sent, 
			Buffered:= Buffered);
	68: MoveLin(Pose := PoseTipSt2,
			ExternalStatecontrol := 0,
			ExternalMove_ID := 0,
			Robot:= Meca500.GVL.Meca500, 
			Error=> Error, 
			Sent:= Sent, 
			Buffered:= Buffered);
	69: MoveLin(Pose := PoseTipSt1,
			ExternalStatecontrol := 0,
			ExternalMove_ID := 0,
			Robot:= Meca500.GVL.Meca500, 
			Error=> Error, 
			Sent:= Sent, 
			Buffered:= Buffered);
	70: MovePose(Pose := PoseMidPose,
			ExternalStatecontrol := 0,
			ExternalMove_ID := 0,
			Robot:= Meca500.GVL.Meca500, 
			Error=> Error, 
			Sent:= Sent, 
			Buffered:= Buffered);	
	71: MoveJoints(Joint_Angle := PoseMotorPlaceTemp,
			ExternalStatecontrol := 0,
			ExternalMove_ID := 0,
			Robot:= Meca500.GVL.Meca500, 
			Error=> Error, 
			Sent:= Sent, 
			Buffered:= Buffered);
	72:	SetCheckpoint(CheckpointID := 209,
			ExternalStatecontrol := 0,
			ExternalMove_ID := 0,
			Robot:= Meca500.GVL.Meca500, 
			Error=> Error, 
			Sent:= Sent, 
			Buffered:= Buffered);
	73: IF Meca500.GVL.Meca500.Inputs.Motion_Status.ReachedCheckPointId = 209 THEN
			stPlcCom.stPlcComOut.bGlueStopValve := FALSE;
			bAllowReCheck := FALSE;
			IF bNeedleDetected THEN
				bReDetectionDone := TRUE;
				bNeedleDetected := FALSE;
				iPositioningStep := 0;
			ELSE
				bDetectionFailed := TRUE;
				bNeedleDetected := FALSE;
				iPositioningStep := 0;
			END_IF
		END_IF 
	100: SetCartLinVel(
			Velocity_Limit := 500,
			ExternalStatecontrol := 0,
			ExternalMove_ID := 0,
			Robot:= Meca500.GVL.Meca500, 
			Error=> Error, 
			Sent:= Sent, 
			Buffered:= Buffered);
	101: MoveLin(Pose := PoseTipSt2,
			ExternalStatecontrol := 0,
			ExternalMove_ID := 0,
			Robot:= Meca500.GVL.Meca500, 
			Error=> Error, 
			Sent:= Sent, 
			Buffered:= Buffered);
	102: MoveLin(Pose := PoseTipSt1,
			ExternalStatecontrol := 0,
			ExternalMove_ID := 0,
			Robot:= Meca500.GVL.Meca500, 
			Error=> Error, 
			Sent:= Sent, 
			Buffered:= Buffered);
	103: MovePose(Pose := PoseMidPose,
			ExternalStatecontrol := 0,
			ExternalMove_ID := 0,
			Robot:= Meca500.GVL.Meca500, 
			Error=> Error, 
			Sent:= Sent, 
			Buffered:= Buffered);	
	104: MoveJoints(Joint_Angle := PoseMotorPlaceTemp,
			ExternalStatecontrol := 0,
			ExternalMove_ID := 0,
			Robot:= Meca500.GVL.Meca500, 
			Error=> Error, 
			Sent:= Sent, 
			Buffered:= Buffered);
			
	105: IF Meca500.GVL.Meca500.Inputs.Motion_Status.ReachedCheckPointId = 220 THEN
			 iPositioningStep := 106;
		END_IF
	106: bDetectionFailed := TRUE;
		iPositioningStep := 0;
		bNeedleFound := FALSE;
END_CASE


IF Sent AND Buffered AND NOT bPassStepSent THEN
	iPositioningStep := iPositioningStep +1;
	Sent := FALSE;
	Buffered := FALSE;
END_IF

METHOD Initialize : BOOL
VAR_INPUT
END_VAR
bDetectionDone := FALSE;
bRobotHomed := FALSE;
bNeedleFound := FALSE;
bReDetectionDone := FALSE;
bDetectionFailed := FALSE;		
bDetectionDone := FALSE;
bReDetectionDone := FALSE;
bAllowReCheck := FALSE;
bNeedleDetected := FALSE;
END_METHOD

END_FUNCTION_BLOCK

// ---- POUs/FB_ASMT60Functions.TcPOU
FUNCTION_BLOCK FB_ASMT60Functions
VAR_INPUT
	bToneEnable				: BOOL;// Toggle to enable tone
	bRedEnable				: BOOL; //Toggle to enable red light
	bYellowEnable			: BOOL; //Toggle to enable yellow light
	bGreenEnable			: BOOL; //Toggle to enable green light
	bBlinkEnable			: BOOL; //Toggle to enable blinking
	tBlinkTime				: TIME := T#500MS; //Adjust blink time
	tToneTime				: TIME :=T#5S;
	tTone2Time				: TIME :=T#500ms;
END_VAR
VAR_OUTPUT
END_VAR
VAR
	BlinkTON				: TON;
	tone5sTON				: TON;
	tone1sTOF				: TOF;
	bBlinkState				: BOOL;
	bToneState				: BOOL;
	bToneTemp				: BOOL;
	bBlink					: BOOL;	
	bRedOut		AT%Q*		: BOOL; //Connect to el2809 Output 13
	bYellowOut	AT%Q*		: BOOL; //Connect to el2809 Output 12
	bGreenOut	AT%Q*		: BOOL; //Connect to el2809 Output 11
	bToneOut	AT%Q*		: BOOL;
	LightCase				: INT;
END_VAR

//////////////////////////////////////////////////////////////////////////////////
//Blinker function
bToneTemp := bToneState;
IF bToneEnable THEN
	tone5sTON(IN:=TRUE, PT:=tToneTime);
	ELSE
	tone1sTOF (IN:=FALSE);
	tone5sTON(IN := FALSE);
    bToneTemp := FALSE;
    bToneState := FALSE;
END_IF

IF tone5sTON.Q THEN
	tone5sTON (IN:=FALSE);
	tone1sTOF(IN := TRUE, PT:=tTone2Time);
	bToneState := NOT bToneState;
END_IF

IF NOT tone5sTON.Q AND tone1sTOF.Q THEN
	tone1sTOF (IN :=FALSE);
END_IF


bBlink := bBlinkState;
IF bBlinkEnable THEN
	BlinkTON(IN :=TRUE, PT :=tBlinkTime);
	IF BlinkTON.Q THEN
		BlinkTON(IN := FALSE);
        bBlinkState := NOT bBlinkState;
	END_IF
ELSE
	BlinkTON(IN := FALSE);
    bBlink := FALSE;
    bBlinkState := FALSE;
END_IF

IF bBlinkEnable AND (bRedEnable OR bYellowEnable OR bGreenEnable) THEN
	LightCase := 10;
	ELSIF bRedEnable OR bYellowEnable OR bGreenEnable THEN
		LightCase := 0;
	ELSIF bToneEnable THEN
		LightCase := 20;
	
END_IF


CASE LightCase OF
0:
//Function for static light
IF bRedEnable THEN
    bRedOut := TRUE; 
    bYellowOut := FALSE;
    bGreenOut := FALSE;
	ELSIF bYellowEnable THEN
  		bRedOut := FALSE;
   		bYellowOut := TRUE; 
    	bGreenOut := FALSE;
	ELSIF bGreenEnable THEN
   		bRedOut := FALSE;
   		bYellowOut := FALSE;
   		bGreenOut := TRUE; 
ELSE
    bRedOut := FALSE;
    bYellowOut := FALSE;
    bGreenOut := FALSE;
END_IF;

10:
//Function for blinking light
IF bRedEnable AND bBlinkEnable THEN
	bRedOut := bBlink;
	bYellowOut := FALSE;
    bGreenOut := FALSE;	
ELSIF bYellowEnable AND bBlinkEnable THEN
	bRedOut := FALSE;
	bYellowOut := bBlink;
	bGreenOut := FALSE;
ELSIF bGreenEnable AND bBlinkEnable THEN
	bRedOut := FALSE;
	bYellowOut := FALSE;
	bGreenOut := bBlink;
END_IF


20:
IF bToneEnable THEN
	bBlinkEnable := TRUE;
	bRedOut := FALSE;
	bGreenOut := FALSE;
	bYellowOut := bBlink;
	bToneOut := tone1sTOF.Q;
ELSE
	bBlinkEnable := FALSE;
	bRedOut := FALSE;
	bGreenOut := FALSE;
	bYellowOut :=FALSE;
	bToneOut := FALSE;
END_IF

END_CASE

END_FUNCTION_BLOCK

// ---- POUs/Sts/Datalog/FB_EventLogger.TcPOU
FUNCTION_BLOCK FB_EventLogger
VAR_INPUT
	bInitDone		: BOOL;
	fbAlarms		: ARRAY [0..18] OF FB_TcAlarm;		// Jokaiselle error tyypille oma fbAlarmi
	bRaiseAlarm		: ARRAY [0..18] OF BOOL;
	bClearAlarm		: ARRAY [0..18] OF BOOL;
	bCondirmAlarm	: ARRAY [0..18] OF BOOL;
	fbSourceInfo	: FB_TcSourceInfo;
	sErrorCode			: STRING;		//Error code tahan
	//fbTest			: reference TO FB_MecaStateMachine;
	stModuleHmi		: REFERENCE TO ST_ModuleHmi;
END_VAR
VAR_OUTPUT
	bErrorActive	:BOOL;
END_VAR
VAR
	//stModuleOut	: reference to ST_ModuleHmi;
	
END_VAR

IF NOT bInitDone THEN
	fbSourceInfo.Clear();
	fbSourceInfo.sName := sErrorCode;		//Strgini variable
	fbAlarms[0].CreateEx(TC_events.ErrorEvent.SafetyCircuitError, TRUE, fbSourceInfo);
	fbAlarms[1].CreateEx(TC_events.ErrorEvent.EstopError, TRUE, fbSourceInfo);
	fbAlarms[2].CreateEx(TC_events.ErrorEvent.PlcSafetyError, TRUE, fbSourceInfo);
	fbAlarms[3].CreateEx(TC_events.ErrorEvent.RobotError, TRUE, fbSourceInfo);
	fbAlarms[4].CreateEx(TC_events.ErrorEvent.LinearAxisHomingError, TRUE, fbSourceInfo);
	fbAlarms[5].CreateEx(TC_events.ErrorEvent.LinearAxisEnableError, TRUE, fbSourceInfo);
	fbAlarms[6].CreateEx(TC_events.ErrorEvent.LinearAxisMovementError, TRUE, fbSourceInfo);
	fbAlarms[7].CreateEx(TC_events.ErrorEvent.StepperMotorError, TRUE, fbSourceInfo);
	fbAlarms[8].CreateEx(TC_events.ErrorEvent.PneumaticError, TRUE, fbSourceInfo);
	fbAlarms[9].CreateEx(TC_events.ErrorEvent.HeaterError, TRUE, fbSourceInfo);
	fbAlarms[10].CreateEx(TC_events.ErrorEvent.HeaterSensorError, TRUE, fbSourceInfo);
	fbAlarms[11].CreateEx(TC_events.ErrorEvent.ImagingError, TRUE, fbSourceInfo);
	fbAlarms[12].CreateEx(TC_events.ErrorEvent.UnderlightDetectionError, TRUE, fbSourceInfo);
	fbAlarms[13].CreateEx(TC_events.ErrorEvent.LaserDetectionError, TRUE, fbSourceInfo);
	fbAlarms[14].CreateEx(TC_events.ErrorEvent.StartupError, TRUE, fbSourceInfo);
	fbAlarms[15].CreateEx(TC_events.ErrorEvent.HatchLockError, TRUE, fbSourceInfo);
	fbAlarms[16].CreateEx(TC_events.ErrorEvent.PalletError, TRUE, fbSourceInfo);
	fbAlarms[17].CreateEx(TC_events.ErrorEvent.NeedleDetectError, TRUE, fbSourceInfo);
	bInitDone := TRUE;
END_IF

IF stModuleHmi.bClearAlarms THEN
	bClearAlarm[0] := TRUE;
	bClearAlarm[1] := TRUE;
	bClearAlarm[2] := TRUE;
	bClearAlarm[3] := TRUE;
	bClearAlarm[4] := TRUE;
	bClearAlarm[5] := TRUE;
	bClearAlarm[6] := TRUE;
	bClearAlarm[7] := TRUE;
	bClearAlarm[8] := TRUE;
	bClearAlarm[9] := TRUE;
	bClearAlarm[10] := TRUE;
	bClearAlarm[11] := TRUE;
	bClearAlarm[12] := TRUE;
	bClearAlarm[13] := TRUE;
	bClearAlarm[14] := TRUE;
	bClearAlarm[15] := TRUE;
	bClearAlarm[16] := TRUE;
	bClearAlarm[17] := TRUE;
END_IF



////////////////////////////////////////////////
IF bRaiseAlarm[0] THEN
	bRaiseAlarm[0] := FALSE;
	fbAlarms[0].ipArguments.Clear().AddString(sErrorCode); //sTest on string variable, tähän voitaisiin kirjottaa vikakoodit suoraan stsActissa. 
	fbAlarms[0].Raise(0);	// 0 määrittää loggeriin tallentuvan ajan, 0 = systime
END_IF

IF bCondirmAlarm[0] THEN
	bCondirmAlarm[0] := FALSE;
	fbAlarms[0].Confirm(0);	 // 0 määrittää loggeriin tallentuvan ajan, 0 = systime
	bClearAlarm[0] := TRUE;
END_IF

IF bClearAlarm[0] THEN
	bClearAlarm[0] := FALSE;
	fbAlarms[0].Clear(0,TRUE);	// 0 määrittää loggeriin tallentuvan ajan, 0 = systime, f/t määrittää voidaanko alarmi confirmata clearauksen jälkeen, falsella voidaan, truella ei. 
							//Falsella ei synny uutta alarmia ennen confirm+clear, truella syntyy pelkällä confirmilla, true ehkä parempio, raise + clear riittää?
END_IF
////////////////////////////////////////////////

IF bRaiseAlarm[1] THEN
	bRaiseAlarm[1] := FALSE;
	fbAlarms[1].ipArguments.Clear().AddString(sErrorCode); //sTest on string variable, tähän voitaisiin kirjottaa vikakoodit suoraan stsActissa. 
	fbAlarms[1].Raise(0);	// 0 määrittää loggeriin tallentuvan ajan, 0 = systime
END_IF

IF bCondirmAlarm[1] THEN
	bCondirmAlarm[1] := FALSE;
	fbAlarms[1].Confirm(0);	 // 0 määrittää loggeriin tallentuvan ajan, 0 = systime
	bClearAlarm[1] := TRUE;
END_IF

IF bClearAlarm[1] THEN
	bClearAlarm[1] := FALSE;
	fbAlarms[1].Clear(0,TRUE);	// 0 määrittää loggeriin tallentuvan ajan, 0 = systime, f/t määrittää voidaanko alarmi confirmata clearauksen jälkeen, falsella voidaan, truella ei. 
							//Falsella ei synny uutta alarmia ennen confirm+clear, truella syntyy pelkällä confirmilla, true ehkä parempio, raise + clear riittää?
END_IF
////////////////////////////////////////////////

IF bRaiseAlarm[2] THEN
	bRaiseAlarm[2] := FALSE;
	fbAlarms[2].ipArguments.Clear().AddString(sErrorCode); //sTest on string variable, tähän voitaisiin kirjottaa vikakoodit suoraan stsActissa. 
	fbAlarms[2].Raise(0);	// 0 määrittää loggeriin tallentuvan ajan, 0 = systime
END_IF

IF bCondirmAlarm[2] THEN
	bCondirmAlarm[2] := FALSE;
	fbAlarms[2].Confirm(0);	 // 0 määrittää loggeriin tallentuvan ajan, 0 = systime
	bClearAlarm[2] := TRUE;
END_IF

IF bClearAlarm[2] THEN
	bClearAlarm[2] := FALSE;
	fbAlarms[2].Clear(0,TRUE);	// 0 määrittää loggeriin tallentuvan ajan, 0 = systime, f/t määrittää voidaanko alarmi confirmata clearauksen jälkeen, falsella voidaan, truella ei. 
							//Falsella ei synny uutta alarmia ennen confirm+clear, truella syntyy pelkällä confirmilla, true ehkä parempio, raise + clear riittää?
END_IF
////////////////////////////////////////////////

IF bRaiseAlarm[3] THEN
	bRaiseAlarm[3] := FALSE;
	fbAlarms[3].ipArguments.Clear().AddString(sErrorCode); //sTest on string variable, tähän voitaisiin kirjottaa vikakoodit suoraan stsActissa. 
	fbAlarms[3].Raise(0);	// 0 määrittää loggeriin tallentuvan ajan, 0 = systime
END_IF

IF bCondirmAlarm[3] THEN
	bCondirmAlarm[3] := FALSE;
	fbAlarms[3].Confirm(0);	 // 0 määrittää loggeriin tallentuvan ajan, 0 = systime
	bClearAlarm[3] := TRUE;
END_IF

IF bClearAlarm[3] THEN
	bClearAlarm[3] := FALSE;
	fbAlarms[3].Clear(0,TRUE);	// 0 määrittää loggeriin tallentuvan ajan, 0 = systime, f/t määrittää voidaanko alarmi confirmata clearauksen jälkeen, falsella voidaan, truella ei. 
							//Falsella ei synny uutta alarmia ennen confirm+clear, truella syntyy pelkällä confirmilla, true ehkä parempio, raise + clear riittää?
END_IF
////////////////////////////////////////////////

IF bRaiseAlarm[4] THEN
	bRaiseAlarm[4] := FALSE;
	fbAlarms[4].ipArguments.Clear().AddString(sErrorCode); //sTest on string variable, tähän voitaisiin kirjottaa vikakoodit suoraan stsActissa. 
	fbAlarms[4].Raise(0);	// 0 määrittää loggeriin tallentuvan ajan, 0 = systime
END_IF

IF bCondirmAlarm[4] THEN
	bCondirmAlarm[4] := FALSE;
	fbAlarms[4].Confirm(0);	 // 0 määrittää loggeriin tallentuvan ajan, 0 = systime
	bClearAlarm[4] := TRUE;
END_IF

IF bClearAlarm[4] THEN
	bClearAlarm[4] := FALSE;
	fbAlarms[4].Clear(0,TRUE);	// 0 määrittää loggeriin tallentuvan ajan, 0 = systime, f/t määrittää voidaanko alarmi confirmata clearauksen jälkeen, falsella voidaan, truella ei. 
							//Falsella ei synny uutta alarmia ennen confirm+clear, truella syntyy pelkällä confirmilla, true ehkä parempio, raise + clear riittää?
END_IF
////////////////////////////////////////////////

IF bRaiseAlarm[5] THEN
	bRaiseAlarm[5] := FALSE;
	fbAlarms[5].ipArguments.Clear().AddString(sErrorCode); //sTest on string variable, tähän voitaisiin kirjottaa vikakoodit suoraan stsActissa. 
	fbAlarms[5].Raise(0);	// 0 määrittää loggeriin tallentuvan ajan, 0 = systime
END_IF

IF bCondirmAlarm[5] THEN
	bCondirmAlarm[5] := FALSE;
	fbAlarms[5].Confirm(0);	 // 0 määrittää loggeriin tallentuvan ajan, 0 = systime
	bClearAlarm[5] := TRUE;
END_IF

IF bClearAlarm[5] THEN
	bClearAlarm[5] := FALSE;
	fbAlarms[5].Clear(0,TRUE);	// 0 määrittää loggeriin tallentuvan ajan, 0 = systime, f/t määrittää voidaanko alarmi confirmata clearauksen jälkeen, falsella voidaan, truella ei. 
							//Falsella ei synny uutta alarmia ennen confirm+clear, truella syntyy pelkällä confirmilla, true ehkä parempio, raise + clear riittää?
END_IF
////////////////////////////////////////////////

IF bRaiseAlarm[6] THEN
	bRaiseAlarm[6] := FALSE;
	fbAlarms[6].ipArguments.Clear().AddString(sErrorCode); //sTest on string variable, tähän voitaisiin kirjottaa vikakoodit suoraan stsActissa. 
	fbAlarms[6].Raise(0);	// 0 määrittää loggeriin tallentuvan ajan, 0 = systime
END_IF

IF bCondirmAlarm[6] THEN
	bCondirmAlarm[6] := FALSE;
	fbAlarms[6].Confirm(0);	 // 0 määrittää loggeriin tallentuvan ajan, 0 = systime
	bClearAlarm[6] := TRUE;
END_IF

IF bClearAlarm[6] THEN
	bClearAlarm[6] := FALSE;
	fbAlarms[6].Clear(0,TRUE);	// 0 määrittää loggeriin tallentuvan ajan, 0 = systime, f/t määrittää voidaanko alarmi confirmata clearauksen jälkeen, falsella voidaan, truella ei. 
							//Falsella ei synny uutta alarmia ennen confirm+clear, truella syntyy pelkällä confirmilla, true ehkä parempio, raise + clear riittää?
END_IF
////////////////////////////////////////////////

IF bRaiseAlarm[7] THEN
	bRaiseAlarm[7] := FALSE;
	fbAlarms[7].ipArguments.Clear().AddString(sErrorCode); //sTest on string variable, tähän voitaisiin kirjottaa vikakoodit suoraan stsActissa. 
	fbAlarms[7].Raise(0);	// 0 määrittää loggeriin tallentuvan ajan, 0 = systime
END_IF

IF bCondirmAlarm[7] THEN
	bCondirmAlarm[7] := FALSE;
	fbAlarms[7].Confirm(0);	 // 0 määrittää loggeriin tallentuvan ajan, 0 = systime
	bClearAlarm[7] := TRUE;
END_IF

IF bClearAlarm[7] THEN
	bClearAlarm[7] := FALSE;
	fbAlarms[7].Clear(0,TRUE);	// 0 määrittää loggeriin tallentuvan ajan, 0 = systime, f/t määrittää voidaanko alarmi confirmata clearauksen jälkeen, falsella voidaan, truella ei. 
							//Falsella ei synny uutta alarmia ennen confirm+clear, truella syntyy pelkällä confirmilla, true ehkä parempio, raise + clear riittää?
END_IF
////////////////////////////////////////////////

IF bRaiseAlarm[8] THEN
	bRaiseAlarm[8] := FALSE;
	fbAlarms[8].ipArguments.Clear().AddString(sErrorCode); //sTest on string variable, tähän voitaisiin kirjottaa vikakoodit suoraan stsActissa. 
	fbAlarms[8].Raise(0);	// 0 määrittää loggeriin tallentuvan ajan, 0 = systime
END_IF

IF bCondirmAlarm[8] THEN
	bCondirmAlarm[8] := FALSE;
	fbAlarms[8].Confirm(0);	 // 0 määrittää loggeriin tallentuvan ajan, 0 = systime
	bClearAlarm[8] := TRUE;
END_IF

IF bClearAlarm[8] THEN
	bClearAlarm[8] := FALSE;
	fbAlarms[8].Clear(0,TRUE);	// 0 määrittää loggeriin tallentuvan ajan, 0 = systime, f/t määrittää voidaanko alarmi confirmata clearauksen jälkeen, falsella voidaan, truella ei. 
							//Falsella ei synny uutta alarmia ennen confirm+clear, truella syntyy pelkällä confirmilla, true ehkä parempio, raise + clear riittää?
END_IF
////////////////////////////////////////////////

IF bRaiseAlarm[9] THEN
	bRaiseAlarm[9] := FALSE;
	fbAlarms[9].ipArguments.Clear().AddString(sErrorCode); //sTest on string variable, tähän voitaisiin kirjottaa vikakoodit suoraan stsActissa. 
	fbAlarms[9].Raise(0);	// 0 määrittää loggeriin tallentuvan ajan, 0 = systime
END_IF

IF bCondirmAlarm[9] THEN
	bCondirmAlarm[9] := FALSE;
	fbAlarms[9].Confirm(0);	 // 0 määrittää loggeriin tallentuvan ajan, 0 = systime
	bClearAlarm[9] := TRUE;
END_IF

IF bClearAlarm[9] THEN
	bClearAlarm[9] := FALSE;
	fbAlarms[9].Clear(0,TRUE);	// 0 määrittää loggeriin tallentuvan ajan, 0 = systime, f/t määrittää voidaanko alarmi confirmata clearauksen jälkeen, falsella voidaan, truella ei. 
							//Falsella ei synny uutta alarmia ennen confirm+clear, truella syntyy pelkällä confirmilla, true ehkä parempio, raise + clear riittää?
END_IF
////////////////////////////////////////////////

IF bRaiseAlarm[10] THEN
	bRaiseAlarm[10] := FALSE;
	fbAlarms[10].ipArguments.Clear().AddString(sErrorCode); //sTest on string variable, tähän voitaisiin kirjottaa vikakoodit suoraan stsActissa. 
	fbAlarms[10].Raise(0);	// 0 määrittää loggeriin tallentuvan ajan, 0 = systime
END_IF

IF bCondirmAlarm[10] THEN
	bCondirmAlarm[10] := FALSE;
	fbAlarms[10].Confirm(0);	 // 0 määrittää loggeriin tallentuvan ajan, 0 = systime
	bClearAlarm[10] := TRUE;
END_IF

IF bClearAlarm[10] THEN
	bClearAlarm[10] := FALSE;
	fbAlarms[10].Clear(0,TRUE);	// 0 määrittää loggeriin tallentuvan ajan, 0 = systime, f/t määrittää voidaanko alarmi confirmata clearauksen jälkeen, falsella voidaan, truella ei. 
							//Falsella ei synny uutta alarmia ennen confirm+clear, truella syntyy pelkällä confirmilla, true ehkä parempio, raise + clear riittää?
END_IF
////////////////////////////////////////////////

IF bRaiseAlarm[11] THEN
	bRaiseAlarm[11] := FALSE;
	fbAlarms[11].ipArguments.Clear().AddString(sErrorCode); //sTest on string variable, tähän voitaisiin kirjottaa vikakoodit suoraan stsActissa. 
	fbAlarms[11].Raise(0);	// 0 määrittää loggeriin tallentuvan ajan, 0 = systime
END_IF

IF bCondirmAlarm[11] THEN
	bCondirmAlarm[11] := FALSE;
	fbAlarms[11].Confirm(0);	 // 0 määrittää loggeriin tallentuvan ajan, 0 = systime
	bClearAlarm[11] := TRUE;
END_IF

IF bClearAlarm[11] THEN
	bClearAlarm[11] := FALSE;
	fbAlarms[11].Clear(0,TRUE);	// 0 määrittää loggeriin tallentuvan ajan, 0 = systime, f/t määrittää voidaanko alarmi confirmata clearauksen jälkeen, falsella voidaan, truella ei. 
							//Falsella ei synny uutta alarmia ennen confirm+clear, truella syntyy pelkällä confirmilla, true ehkä parempio, raise + clear riittää?
END_IF
////////////////////////////////////////////////

IF bRaiseAlarm[12] THEN
	bRaiseAlarm[12] := FALSE;
	fbAlarms[12].ipArguments.Clear().AddString(sErrorCode); //sTest on string variable, tähän voitaisiin kirjottaa vikakoodit suoraan stsActissa. 
	fbAlarms[12].Raise(0);	// 0 määrittää loggeriin tallentuvan ajan, 0 = systime
END_IF

IF bCondirmAlarm[12] THEN
	bCondirmAlarm[12] := FALSE;
	fbAlarms[12].Confirm(0);	 // 0 määrittää loggeriin tallentuvan ajan, 0 = systime
	bClearAlarm[12] := TRUE;
END_IF

IF bClearAlarm[12] THEN
	bClearAlarm[12] := FALSE;
	fbAlarms[12].Clear(0,TRUE);	// 0 määrittää loggeriin tallentuvan ajan, 0 = systime, f/t määrittää voidaanko alarmi confirmata clearauksen jälkeen, falsella voidaan, truella ei. 
							//Falsella ei synny uutta alarmia ennen confirm+clear, truella syntyy pelkällä confirmilla, true ehkä parempio, raise + clear riittää?
END_IF
////////////////////////////////////////////////

IF bRaiseAlarm[13] THEN
	bRaiseAlarm[13] := FALSE;
	fbAlarms[13].ipArguments.Clear().AddString(sErrorCode); //sTest on string variable, tähän voitaisiin kirjottaa vikakoodit suoraan stsActissa. 
	fbAlarms[13].Raise(0);	// 0 määrittää loggeriin tallentuvan ajan, 0 = systime
END_IF

IF bCondirmAlarm[13] THEN
	bCondirmAlarm[13] := FALSE;
	fbAlarms[13].Confirm(0);	 // 0 määrittää loggeriin tallentuvan ajan, 0 = systime
	bClearAlarm[13] := TRUE;
END_IF

IF bClearAlarm[13] THEN
	bClearAlarm[13] := FALSE;
	fbAlarms[13].Clear(0,TRUE);	// 0 määrittää loggeriin tallentuvan ajan, 0 = systime, f/t määrittää voidaanko alarmi confirmata clearauksen jälkeen, falsella voidaan, truella ei. 
							//Falsella ei synny uutta alarmia ennen confirm+clear, truella syntyy pelkällä confirmilla, true ehkä parempio, raise + clear riittää?
END_IF
////////////////////////////////////////////////

IF bRaiseAlarm[14] THEN
	bRaiseAlarm[14] := FALSE;
	fbAlarms[14].ipArguments.Clear().AddString(sErrorCode); //sTest on string variable, tähän voitaisiin kirjottaa vikakoodit suoraan stsActissa. 
	fbAlarms[14].Raise(0);	// 0 määrittää loggeriin tallentuvan ajan, 0 = systime
END_IF

IF bCondirmAlarm[14] THEN
	bCondirmAlarm[14] := FALSE;
	fbAlarms[14].Confirm(0);	 // 0 määrittää loggeriin tallentuvan ajan, 0 = systime
	bClearAlarm[14] := TRUE;
END_IF

IF bClearAlarm[14] THEN
	bClearAlarm[14] := FALSE;
	fbAlarms[14].Clear(0,TRUE);	// 0 määrittää loggeriin tallentuvan ajan, 0 = systime, f/t määrittää voidaanko alarmi confirmata clearauksen jälkeen, falsella voidaan, truella ei. 
							//Falsella ei synny uutta alarmia ennen confirm+clear, truella syntyy pelkällä confirmilla, true ehkä parempio, raise + clear riittää?
END_IF
////////////////////////////////////////////////

IF bRaiseAlarm[15] THEN
	bRaiseAlarm[15] := FALSE;
	fbAlarms[15].ipArguments.Clear().AddString(sErrorCode); //sTest on string variable, tähän voitaisiin kirjottaa vikakoodit suoraan stsActissa. 
	fbAlarms[15].Raise(0);	// 0 määrittää loggeriin tallentuvan ajan, 0 = systime
END_IF

IF bCondirmAlarm[15] THEN
	bCondirmAlarm[15] := FALSE;
	fbAlarms[15].Confirm(0);	 // 0 määrittää loggeriin tallentuvan ajan, 0 = systime
	bClearAlarm[15] := TRUE;
END_IF

IF bClearAlarm[15] THEN
	bClearAlarm[15] := FALSE;
	fbAlarms[15].Clear(0,TRUE);	// 0 määrittää loggeriin tallentuvan ajan, 0 = systime, f/t määrittää voidaanko alarmi confirmata clearauksen jälkeen, falsella voidaan, truella ei. 
							//Falsella ei synny uutta alarmia ennen confirm+clear, truella syntyy pelkällä confirmilla, true ehkä parempio, raise + clear riittää?
END_IF
////////////////////////////////////////////////

IF bRaiseAlarm[16] THEN
	bRaiseAlarm[16] := FALSE;
	fbAlarms[16].ipArguments.Clear().AddString(sErrorCode); //sTest on string variable, tähän voitaisiin kirjottaa vikakoodit suoraan stsActissa. 
	fbAlarms[16].Raise(0);	// 0 määrittää loggeriin tallentuvan ajan, 0 = systime
END_IF

IF bCondirmAlarm[16] THEN
	bCondirmAlarm[16] := FALSE;
	fbAlarms[16].Confirm(0);	 // 0 määrittää loggeriin tallentuvan ajan, 0 = systime
	bClearAlarm[16] := TRUE;
END_IF

IF bClearAlarm[16] THEN
	bClearAlarm[16] := FALSE;
	fbAlarms[16].Clear(0,TRUE);	// 0 määrittää loggeriin tallentuvan ajan, 0 = systime, f/t määrittää voidaanko alarmi confirmata clearauksen jälkeen, falsella voidaan, truella ei. 
							//Falsella ei synny uutta alarmia ennen confirm+clear, truella syntyy pelkällä confirmilla, true ehkä parempio, raise + clear riittää?
END_IF
////////////////////////////////////////////////

IF bRaiseAlarm[17] THEN
	bRaiseAlarm[17] := FALSE;
	fbAlarms[17].ipArguments.Clear().AddString(sErrorCode); //sTest on string variable, tähän voitaisiin kirjottaa vikakoodit suoraan stsActissa. 
	fbAlarms[17].Raise(0);	// 0 määrittää loggeriin tallentuvan ajan, 0 = systime
END_IF

IF bCondirmAlarm[17] THEN
	bCondirmAlarm[17] := FALSE;
	fbAlarms[17].Confirm(0);	 // 0 määrittää loggeriin tallentuvan ajan, 0 = systime
	bClearAlarm[17] := TRUE;
END_IF

IF bClearAlarm[17] THEN
	bClearAlarm[17] := FALSE;
	fbAlarms[17].Clear(0,TRUE);	// 0 määrittää loggeriin tallentuvan ajan, 0 = systime, f/t määrittää voidaanko alarmi confirmata clearauksen jälkeen, falsella voidaan, truella ei. 
							//Falsella ei synny uutta alarmia ennen confirm+clear, truella syntyy pelkällä confirmilla, true ehkä parempio, raise + clear riittää?
END_IF
////////////////////////////////////////////////
IF fbAlarms[0].bActive OR fbAlarms[1].bActive OR fbAlarms[2].bActive OR fbAlarms[3].bActive OR fbAlarms[4].bActive OR fbAlarms[5].bActive OR fbAlarms[6].bActive OR fbAlarms[7].bActive OR fbAlarms[8].bActive OR fbAlarms[9].bActive OR fbAlarms[10].bActive OR fbAlarms[11].bActive OR fbAlarms[12].bActive OR fbAlarms[13].bActive OR fbAlarms[14].bActive OR fbAlarms[15].bActive OR fbAlarms[16].bActive OR fbAlarms[17].bActive THEN
	bErrorActive := TRUE;
	ELSE
		bErrorActive := FALSE;
END_IF

END_FUNCTION_BLOCK

// ---- POUs/Sts/Com/FB_RecipeDataExchange.TcPOU
FUNCTION_BLOCK FB_RecipeDataExchange
VAR_INPUT
	trigAdsWrite		: BOOL;
	sendRecipeData	: REFERENCE TO ST_Recipes; // Kirjoittaa nämä tiedot -> toisen pc: MAIN.reveicedLaserData
	stModuleHmi			: REFERENCE TO ST_ModuleHmi;
END_VAR
VAR_OUTPUT
END_VAR
VAR
	adsWriteStatus : INT :=0;

	fbAdsWriteRecipe		:FB_WriteAdsSymByName :=(
		sNetId :='192.168.1.10.1.1',
		nPort := 852,
		eComMode :=E_AdsComMode.eAdsComModeFastCom,
		tTimeout :=DEFAULT_ADS_TIMEOUT);
	bStart		: BOOL;
	delayedStart	:TON;
	resetCounter	:INT :=0;
	bAllowStart		:BOOL;
	retryDelayTON	:TON;
	bRetrytimer		:BOOL :=FALSE;
END_VAR


delayedStart (IN:=TRUE, PT:=T#10S);
bAllowStart := TRUE;
IF stModuleHmi.bResetCommunication THEN
	adsWriteStatus := 30;
END_IF

CASE adsWriteStatus OF

0 : 
		IF NOT fbAdsWriteRecipe.bBusy  AND delayedStart.Q AND bAllowStart THEN	// oli trigAdsWrite
			//trigAdsWrite := FALSE; //Dsable this maybe, so that data transfers continuously
			adsWriteStatus := 10;
		END_IF
10 :

		fbAdsWriteRecipe(bWrite := FALSE);
		fbAdsWriteRecipe(
			sVarName := 'MAIN_VISION.ReceivedRecipeData', //Destination symbol name/location
			nLen := SIZEOF(sendRecipeData), //Lähetettävän tiedon koko saadaan suoraan structuurista
			nSrcAddr := ADR(sendRecipeData), 	//Lähetettävän tiedon osoite saadaan suoraan structuurista
			bWrite := TRUE );
		adsWriteStatus := 20;
20 :

		fbAdsWriteRecipe(bWrite := FALSE);
		IF NOT fbAdsWriteRecipe.bBusy THEN
			IF NOT fbAdsWriteRecipe.bError THEN
				adsWriteStatus := 0;
			ELSE
				adsWriteStatus := 30;
			END_IF
		END_IF
30 :
 	IF NOT bRetryTimer THEN
        retryDelayTON(IN := TRUE, PT := T#10S);
        bRetrytimer := TRUE;
    ELSE
        retryDelayTON(IN := TRUE); // keep running
    END_IF

		IF retryDelayTON.Q THEN
        	retryDelayTON(IN := FALSE); // Reset timer 
        	bRetrytimer := FALSE;

        	IF delayedStart.Q AND resetCounter < 3 AND bAllowStart THEN
            	resetCounter := resetCounter + 1;
            	adsWriteStatus := 10;         // retry write
        	ELSE
            	bAllowStart := FALSE;         // 3 attempts failed
            	adsWriteStatus := 0;          // go idle?
        END_IF
    END_IF
END_CASE

END_FUNCTION_BLOCK

